IF month > 2 THEN
	count := (month - 1) * 30;
	IF month > 7 THEN count := count + SHR(month - 3,1); ELSE count := count + SHR(month - 4,1); END_IF;
	(* chech for leap year and add one day if true *)
	IF SHL(year,14) = 0 THEN count := count + 1; END_IF;
ELSE
	count := (month - 1) * 31;
END_IF;


SetDataTime := DWORD_TO_DT(DATE_TO_DWORD( DWORD_TO_DATE((INT_TO_DWORD(count + day - 1) + SHR(INT_TO_DWORD(year) * 1461 - 2878169, 2)) * 86400))
				+ INT_TO_DWORD(SECOND)
				+ INT_TO_DWORD(MINUTE) * 60
				+ INT_TO_DWORD(HOUR) * 3600);
END_FUNCTION

(* POU Plant/SYS_Proc, ST *)
PROGRAM SYS_Proc
VAR
	fALARM_PB		:FLT_TAP;
	fALARM_TB		:FLT_TAP;
	fALARM_PM		:FLT_TAP;
	fALARM_ALARM_PM_PB_TB		:FLT_TAP;

(*	fGZB_ST			:FLT_TAP;  (* GATEWAY ZIGBEE *)*)
	fVPN_ST1		:FLT_TAP;  (* VPN CONNECT *)
	fVPN_ST2		:FLT_TAP;  (* VPN STATUS *)
	fKEY_CT_ST		:FLT_TAP;  (* DOOR1 *)
	fKEY_SCT_ST		:FLT_TAP;  (* DOOR2 *)
	fKEY_QE_ST		:FLT_TAP;  (* DOOR3 *)


	fBostAttivo	:FLT_TAP;

	fALARM_MancatoRaggiungimentoAcqua		:FLT_TAP;
	DelayfALARM_MancatoRaggiungimentoAcqua:TON;

	pio: BOOL;
END_VAR
(*************** ISPESL *****************)
(*
fALARM_PB(IN:=ALARM_PB);
IF fALARM_PB.EVH THEN
	LogEv(EL_AlarmStop,EO_PBV,1,1,'Over_Pressure_Alarm');
END_IF

fALARM_TB(IN:=ALARM_TB);
IF fALARM_TB.EVH THEN
	LogEv(EL_AlarmStop,EO_TBV,1,1,'Over_Temperature_Alarm');
END_IF

fALARM_PM(IN:=ALARM_PM);
IF fALARM_PM.EVH THEN
	LogEv(EL_AlarmStop,EO_PMV,1,1,'Under_Pressure_Alarm');
END_IF
*)
(*
fALARM_ALARM_PM_PB_TB(IN:=ALARM_PM_PB_TB);
IF fALARM_ALARM_PM_PB_TB.EVH THEN
	LogEv(EL_AlarmStop,EO_PMV,1,1,'Allarmi_ISPESL');
END_IF
*)

(*



(****************************************)

(*### VPN Connection Check ###*)
fVPN_ST1(IN:=VPN_ST1);
IF fVPN_ST1.EVH THEN
	LogEv(EL_Log,EO_VPN,1,1,'CONNECT_ON');
END_IF
IF fVPN_ST1.EVL THEN
	LogEv(EL_Log,EO_VPN,1,2,'CONNECT_OFF');
END_IF
(*
(*### VPN Status Check ###*)
fVPN_ST2(IN:=VPN_ST2);
IF fVPN_ST2.EVH THEN
	LogEv(EL_Log,EO_VPN,1,3,'STATUS_UP');
END_IF
IF fVPN_ST2.EVL THEN
	LogEv(EL_Wrn,EO_VPN,1,4,'STATUS_DOWN');
END_IF

(*### DOOR01 Status Check ###*)
fKEY_CT_ST(IN:=KEY_CT_ST);
IF fKEY_CT_ST.EVH THEN
	LogEv(EL_Log,EO_DOOR,1,2,'Centrale_termica_Close');
END_IF
IF fKEY_CT_ST.EVL THEN
	LogEv(EL_Wrn,EO_DOOR,1,1,'Centrale_termica_Open');
END_IF

(*### DOOR02 Status Check ###*)
fKEY_SCT_ST(IN:=KEY_SCT_ST);
IF fKEY_SCT_ST.EVH THEN
	LogEv(EL_Log,EO_DOOR,2,2,'Sottocentrale_termica_Close');
END_IF
IF fKEY_SCT_ST.EVL THEN
	LogEv(EL_Wrn,EO_DOOR,2,1,'Sottocentrale_termica_Open');
END_IF
*)
(*### DOOR03 Status Check ###*)
fKEY_QE_ST(IN:=KEY_QE_ST);
IF fKEY_QE_ST.EVH THEN
	LogEv(EL_Log,EO_DOOR,3,2,'Quadro_Close');
END_IF
IF fKEY_QE_ST.EVL THEN
	LogEv(EL_Wrn,EO_DOOR,3,1,'Quadro_Open');
END_IF

*)

pio:=FALSE;
END_PROGRAM

(* POU Utils Functions/FLT_TAP, ST *)
FUNCTION_BLOCK FLT_TAP
VAR_INPUT
	IN		: BOOL;
	TAP		: BYTE:=4;
	INITEV	: BOOL:=TRUE;
END_VAR
VAR_OUTPUT
	OUT		: BOOL;
	EVH		: BOOL;
	EVL		: BOOL;
END_VAR
VAR
	init	: BOOL:=FALSE;
	cnt		: BYTE;
END_VAR
EVH:=FALSE;
EVL:=FALSE;

IF NOT init THEN
	init := TRUE;
	IF INITEV THEN
		OUT  := NOT IN;
		cnt  := TAP;
	ELSE
		OUT  := IN;
	END_IF
END_IF

IF OUT<>IN THEN
	cnt:=cnt+1;
	IF cnt>TAP THEN
		OUT:=IN;
		cnt:=0;
		IF OUT THEN EVH:=TRUE; ELSE EVL:=TRUE; END_IF
	END_IF
ELSE
	cnt:=0;
END_IF
END_FUNCTION_BLOCK

(* POU Utils/USRLED_Update, ST *)
PROGRAM USRLED_Update
VAR
	OldStatus: en_SYS_Status;

	aFS : ARRAY [0..24] OF FLASHING_SEQUENCE :=
		(Colour:=GREEN,  Frequency:=1,   Relation:=128, Duration:=t#0s,    NextIndex:=0),  (* 0 => RUNNING *)
		(Colour:=ORANGE, Frequency:=1,   Relation:=128, Duration:=t#0s,    NextIndex:=1),  (* 1 => INIT *)
		(Colour:=RED,    Frequency:=4,   Relation:=128, Duration:=t#0s,    NextIndex:=2),  (* 2 => ERROR *)
		(Colour:=RED,    Frequency:=10,  Relation:=128, Duration:=t#0s,    NextIndex:=3),  (* 3 => ALARM *)
		(Colour:=ORANGE, Frequency:=200, Relation:=16,  Duration:=t#100ms, NextIndex:=11), (* 10 *)
		(Colour:=ORANGE, Frequency:=200, Relation:=32,  Duration:=t#100ms, NextIndex:=12),
		(Colour:=ORANGE, Frequency:=200, Relation:=64,  Duration:=t#100ms, NextIndex:=13),
		(Colour:=ORANGE, Frequency:=200, Relation:=128, Duration:=t#100ms, NextIndex:=14),
		(Colour:=ORANGE, Frequency:=200, Relation:=192, Duration:=t#100ms, NextIndex:=15),
		(Colour:=ORANGE, Frequency:=200, Relation:=128, Duration:=t#100ms, NextIndex:=16),
		(Colour:=ORANGE, Frequency:=200, Relation:=64,  Duration:=t#100ms, NextIndex:=17),
		(Colour:=ORANGE, Frequency:=200, Relation:=32,  Duration:=t#100ms, NextIndex:=18),
		(Colour:=ORANGE, Frequency:=200, Relation:=16,  Duration:=t#100ms, NextIndex:=19),
		(Colour:=ORANGE, Frequency:=200, Relation:=8,   Duration:=t#100ms, NextIndex:=10),
		(Colour:=GREEN,  Frequency:=200, Relation:=16,  Duration:=t#100ms, NextIndex:=21), (* 20 *)
		(Colour:=GREEN,  Frequency:=200, Relation:=32,  Duration:=t#100ms, NextIndex:=22),
		(Colour:=GREEN,  Frequency:=200, Relation:=64,  Duration:=t#100ms, NextIndex:=23),
		(Colour:=GREEN,  Frequency:=200, Relation:=128, Duration:=t#100ms, NextIndex:=24),
		(Colour:=GREEN,  Frequency:=200, Relation:=192, Duration:=t#100ms, NextIndex:=25),
		(Colour:=GREEN,  Frequency:=200, Relation:=128, Duration:=t#100ms, NextIndex:=26),
		(Colour:=GREEN,  Frequency:=200, Relation:=64,  Duration:=t#100ms, NextIndex:=27),
		(Colour:=GREEN,  Frequency:=200, Relation:=32,  Duration:=t#100ms, NextIndex:=28),
		(Colour:=GREEN,  Frequency:=200, Relation:=16,  Duration:=t#100ms, NextIndex:=29),
		(Colour:=GREEN,  Frequency:=200, Relation:=8,   Duration:=t#100ms, NextIndex:=20);

	pFS : POINTER TO FLASHING_SEQUENCE;


END_VAR
IF Sys.Status <> OldStatus THEN

	OldStatus:=Sys.Status;

	CASE OldStatus OF

		S_STARTUP:
			pFS:=ADR(aFS);
			SET_FLASHING_SEQUENCE(EN:=TRUE, POINTER_TO_POINTER_TO_ARRAY:=ADR(pFS));
			SET_FLASHING_SEQUENCE_INDEX(EN:=TRUE, IMMEDIATE:=FALSE, INDEX:=1);
			START_FLASHING_SEQUENCE(EN:=TRUE);

		S_RUNNING:
			SET_FLASHING_SEQUENCE_INDEX(EN:=TRUE, IMMEDIATE:=TRUE, INDEX:=0);

	END_CASE

END_IF
END_PROGRAM

(* POU Utils Functions/AVERAGE_T, ST *)
FUNCTION_BLOCK AVERAGE_T
VAR_INPUT
	IN: 	INT;
END_VAR
VAR_OUTPUT
	HI:		INT;
	AVG:	INT;
	LOW:	INT;
	ERR:	BOOL;
END_VAR
VAR
	sum:	DINT;
	cnt:	WORD;
END_VAR
IF cnt>=65000 THEN
	ERR:=TRUE;
	Read();
	sum := sum - AVG;
	cnt := cnt + 1;
END_IF

sum := sum + IN;
cnt := cnt + 1;

IF IN<LOW THEN  LOW:=IN; END_IF
IF IN>HI  THEN HI :=IN; END_IF
END_FUNCTION_BLOCK
ACTION Read:
AVG := DINT_TO_INT(sum/cnt);
END_ACTION
ACTION Reset:
HI:=IN;
AVG:=IN;
LOW:=IN;
ERR:=FALSE;

sum:=IN;
cnt:=1;
END_ACTION

(* POU Utils Functions/COPY_32SWAP16, ST *)
FUNCTION COPY_32SWAP16:BOOL
VAR_INPUT
	pSourceAddress		:POINTER TO ARRAY[1..2] OF WORD;
	pDestinationAddress	:POINTER TO ARRAY[1..2] OF WORD;
END_VAR
VAR
END_VAR
pDestinationAddress^[1]:=pSourceAddress^[2];
pDestinationAddress^[2]:=pSourceAddress^[1];
END_FUNCTION

(* POU Utils Functions/FLT_EVENT, ST *)
FUNCTION_BLOCK FLT_EVENT
VAR_INPUT
	IN		: BOOL;
	INITEV	: BOOL:=TRUE;
END_VAR
VAR_OUTPUT
	EVH		: BOOL;
	EVL		: BOOL;
END_VAR
VAR
	init	: BOOL:=FALSE;
	old		: BOOL;
END_VAR
EVH:=FALSE;
EVL:=FALSE;

IF NOT init THEN
	init:=TRUE;
	IF INITEV THEN
		old := NOT IN;
	ELSE
		old := IN;
	END_IF
END_IF

IF old<>IN THEN
	old:=IN;
	IF IN THEN EVH:=TRUE; ELSE EVL:=TRUE; END_IF
END_IF
END_FUNCTION_BLOCK

(* POU Utils Functions/FLT_TIME, ST *)
FUNCTION_BLOCK FLT_TIME
VAR_INPUT
	IN		: BOOL;
	TTAP	: TIME:=T#5s;
	INITEV	: BOOL:=TRUE;
END_VAR
VAR_OUTPUT
	OUT		: BOOL;
	EVH		: BOOL;
	EVL		: BOOL;
END_VAR
VAR
	init	: BOOL:=FALSE;
	timer	: TON;
END_VAR
EVH:=FALSE;
EVL:=FALSE;

IF NOT init THEN
	init := TRUE;
	IF INITEV THEN
		OUT  := NOT IN;
	ELSE
		OUT  := IN;
	END_IF
END_IF

IF OUT<>IN THEN
	timer(IN:=TRUE,PT:=TTAP);
	IF timer.Q THEN
		OUT:=IN;
		timer(IN:=FALSE);
		IF OUT THEN EVH:=TRUE; ELSE EVL:=TRUE; END_IF
	END_IF
ELSE
	timer(IN:=FALSE);
END_IF
END_FUNCTION_BLOCK

(* POU Utils Functions/FUN_2Word_to_REAL, ST *)
FUNCTION FUN_2Word_to_REAL : REAL
VAR_INPUT

	WORDH:WORD;
	WORDL:WORD;
	Decimali:INT;
	signed:BOOL;     (* false unsigned - true signed *)

END_VAR

VAR

	ValoreDWord: DWORD;
	ValoreDint: DINT;
	testINT1: DINT;
	testINT2: DINT;


END_VAR
IF signed THEN

		(* Stabilisco il segno della variabile letta *)

		IF WORDH> 16#8000 THEN
			ValoreDint:=((16#FFFFFFFF-(WORDH*65535+WORDL)))*(-1);
		ELSE
			ValoreDint:=(WORDH*65535+WORDL);
		END_IF;

	CASE Decimali OF
		0 : FUN_2Word_to_REAL:=DINT_TO_REAL (ValoreDint);
		1 : FUN_2Word_to_REAL:=DINT_TO_REAL (ValoreDint)/10;
		2 : FUN_2Word_to_REAL:=DINT_TO_REAL (ValoreDint)/100;
		3 : FUN_2Word_to_REAL:=DINT_TO_REAL (ValoreDint)/1000;
		4 : FUN_2Word_to_REAL:=DINT_TO_REAL (ValoreDint)/10000;
		5 : FUN_2Word_to_REAL:=DINT_TO_REAL (ValoreDint)/100000;
		6 : FUN_2Word_to_REAL:=DINT_TO_REAL (ValoreDint)/1000000;
	END_CASE;


ELSE
	ValoreDWord:=(WORDH*65535+WORDL);

	CASE Decimali OF
		0 : FUN_2Word_to_REAL:=DWORD_TO_REAL (ValoreDWord);
		1 : FUN_2Word_to_REAL:=DWORD_TO_REAL (ValoreDWord)/10;
		2 : FUN_2Word_to_REAL:=DWORD_TO_REAL (ValoreDWord)/100;
		3 : FUN_2Word_to_REAL:=DWORD_TO_REAL (ValoreDWord)/1000;
		4 : FUN_2Word_to_REAL:=DWORD_TO_REAL (ValoreDWord)/10000;
		5 : FUN_2Word_to_REAL:=DWORD_TO_REAL (ValoreDWord)/100000;
		6 : FUN_2Word_to_REAL:=DWORD_TO_REAL (ValoreDWord)/1000000;
	END_CASE;
END_IF;
END_FUNCTION

(* POU Utils/FUN_ByteAsci, ST *)
FUNCTION FUN_ByteAsci : STRING(1)
VAR_INPUT
	ByteIn:BYTE;
END_VAR
VAR
END_VAR
CASE ByteIn OF

	32: FUN_ByteAsci:=' ';
	33: FUN_ByteAsci:='!';
	34: FUN_ByteAsci:='"';
	35: FUN_ByteAsci:='#';

	37: FUN_ByteAsci:='%';
	38: FUN_ByteAsci:='&';

	40: FUN_ByteAsci:='(';
	41: FUN_ByteAsci:=')';
	42: FUN_ByteAsci:='*';
	43: FUN_ByteAsci:='+';
	44: FUN_ByteAsci:=',';
	45: FUN_ByteAsci:='-';
	46: FUN_ByteAsci:='.';
	47: FUN_ByteAsci:='/';
	48: FUN_ByteAsci:='0';
	49: FUN_ByteAsci:='1';
	50: FUN_ByteAsci:='2';
	51: FUN_ByteAsci:='3';
	52: FUN_ByteAsci:='4';
	53: FUN_ByteAsci:='5';
	54: FUN_ByteAsci:='6';
	55: FUN_ByteAsci:='7';
	56: FUN_ByteAsci:='8';
	57: FUN_ByteAsci:='9';
	58: FUN_ByteAsci:=':';
	59: FUN_ByteAsci:=';';
	60: FUN_ByteAsci:='<';
	61: FUN_ByteAsci:='=';
	62: FUN_ByteAsci:='>';
	63: FUN_ByteAsci:='?';
	64: FUN_ByteAsci:='@';
	65: FUN_ByteAsci:='A';
	66: FUN_ByteAsci:='B';
	67: FUN_ByteAsci:='C';
	68: FUN_ByteAsci:='D';
	69: FUN_ByteAsci:='E';
	70: FUN_ByteAsci:='F';
	71: FUN_ByteAsci:='G';
	72: FUN_ByteAsci:='H';
	73: FUN_ByteAsci:='I';
	74: FUN_ByteAsci:='J';
	75: FUN_ByteAsci:='K';
	76: FUN_ByteAsci:='L';
	77: FUN_ByteAsci:='M';
	78: FUN_ByteAsci:='N';
	79: FUN_ByteAsci:='O';
	80: FUN_ByteAsci:='P';
	81: FUN_ByteAsci:='Q';
	82: FUN_ByteAsci:='R';
	83: FUN_ByteAsci:='S';
	84: FUN_ByteAsci:='T';
	85: FUN_ByteAsci:='U';
	86: FUN_ByteAsci:='V';
	87: FUN_ByteAsci:='W';
	88: FUN_ByteAsci:='X';
	89: FUN_ByteAsci:='Y';
	90: FUN_ByteAsci:='Z';
	91: FUN_ByteAsci:='[';
	92: FUN_ByteAsci:='\';
	93: FUN_ByteAsci:=']';
	94: FUN_ByteAsci:='^';
	95: FUN_ByteAsci:='_';
	96: FUN_ByteAsci:='`';
	97: FUN_ByteAsci:='a';
	98: FUN_ByteAsci:='b';
	99: FUN_ByteAsci:='c';
	100: FUN_ByteAsci:='d';
	101: FUN_ByteAsci:='e';
	102: FUN_ByteAsci:='f';
	103: FUN_ByteAsci:='g';
	104: FUN_ByteAsci:='h';
	105: FUN_ByteAsci:='i';
	106: FUN_ByteAsci:='j';
	107: FUN_ByteAsci:='k';
	108: FUN_ByteAsci:='l';
	109: FUN_ByteAsci:='m';
	110: FUN_ByteAsci:='n';
	111: FUN_ByteAsci:='o';
	112: FUN_ByteAsci:='p';
	113: FUN_ByteAsci:='q';
	114: FUN_ByteAsci:='r';
	115: FUN_ByteAsci:='s';
	116: FUN_ByteAsci:='t';
	117: FUN_ByteAsci:='u';
	118: FUN_ByteAsci:='v';
	119: FUN_ByteAsci:='w';
	120: FUN_ByteAsci:='x';
	121: FUN_ByteAsci:='y';
	122: FUN_ByteAsci:='z';
	123: FUN_ByteAsci:='{';
	124: FUN_ByteAsci:='|';
	125: FUN_ByteAsci:='}';
	126: FUN_ByteAsci:='~';

	167: FUN_ByteAsci:='°';
	176: FUN_ByteAsci:='°';


ELSE
	FUN_ByteAsci:='';

END_CASE
END_FUNCTION

(* POU Utils Functions/FUN_DEAD_ZONE, ST *)
FUNCTION FUN_DEAD_ZONE : INT
VAR_INPUT
	X : INT;
	L : INT;
END_VAR
VAR
	DEAD_BAND: BOOL;
END_VAR
IF X>=FUN_DEAD_ZONE+L THEN
	FUN_DEAD_ZONE := X ;
ELSIF X <= FUN_DEAD_ZONE-L THEN
	FUN_DEAD_ZONE := X;
ELSE
	FUN_DEAD_ZONE :=FUN_DEAD_ZONE;
END_IF;
END_FUNCTION

(* POU Utils Functions/LAMP_AL_GENERALE, ST *)
FUNCTION_BLOCK LAMP_AL_GENERALE
VAR_INPUT

	Allarme: BOOL;
	Warning: BOOL;
END_VAR
VAR_OUTPUT
	SistemaOK:BOOL;
	SistemaInAllarme:BOOL;
	SistemaWarning:BOOL;
	AllarmeLampada:BOOL;
END_VAR
VAR
	Lampeggio:BLINK;
END_VAR
IF Allarme THEN       					(* Se Allarme Attivo Lucde fissa ON *)
	SistemaInAllarme:=TRUE;
	SistemaWarning:=FALSE;
	AllarmeLampada:=TRUE;
ELSIF Warning THEN					(* Se Allarme Attivo Lucde fissa pulse *)
	SistemaInAllarme:=FALSE;
	SistemaWarning:=TRUE;
	Lampeggio(ENABLE:=TRUE , TIMELOW:=t#1s , TIMEHIGH:=t#1s , OUT=>AllarmeLampada );
ELSE
	SistemaInAllarme:=FALSE;
	SistemaWarning:=FALSE;
	AllarmeLampada:=FALSE;
END_IF
END_FUNCTION_BLOCK

(* POU Utils Functions/LINEAR_BAD, ST *)
FUNCTION LINEAR_BAD : INT (* Linear interpolation *)
VAR_INPUT
	PuntoMinX	: INT;
	PuntoMaxX	: INT;
	ValIn		: INT;
	PuntoMinY	: REAL;
	PuntoMaxY	: REAL;
	Decimali	: BYTE;
END_VAR
VAR
	Gain				: REAL;
	PuntoMinX_R			: REAL;
	PuntoMaxX_R			: REAL;
	Linearizzazione_R	: REAL;
END_VAR
PuntoMinX_R:=INT_TO_REAL(PuntoMinX);
PuntoMaxX_R:=INT_TO_REAL(PuntoMaxX);

Gain:=(PuntoMaxX_R-PuntoMinX_R)/(PuntoMaxY-PuntoMinY);	(* Calcolo in guadagno per la linarizzazione *)
Linearizzazione_R:=PuntoMinx+(Gain*(ValIn-PuntoMinY));	(* Ottengo il valore linearizzato *)

LINEAR_BAD:=REAL_TO_INT(Linearizzazione_R*(EXPT(10, Decimali)));  (* Ottengo intero con i decimai voluti *)
END_FUNCTION

(* POU Utils Functions/MEMCLR, ST *)
FUNCTION MEMCLR:BOOL
VAR_INPUT
	pDestinationAddress:POINTER TO ARRAY[1..2] OF BYTE;
	BytesToClear:WORD;
END_VAR
VAR
END_VAR
WHILE (BytesToClear > 0) DO
	pDestinationAddress^[1]:=0;
	pDestinationAddress:=ADR(pDestinationAddress^[2]); (* increment destination *)
	BytesToClear:=BytesToClear -1; (* decrement number of bytes to copy *)
END_WHILE
END_FUNCTION

(* POU Plant_Objects/obj_AI_GEN, ST *)
FUNCTION_BLOCK obj_AI_GEN
(* === TEMPERATURE PROBE FROM ANALOG INPUT ===
   v1.0[16/04/05] - Versioning
*)
VAR_INPUT
	(* Settings *)
	ID				: BYTE;
	PuntoMinX		: INT;			(* Parametri per la scalatura *)
	PuntoMaxX		: INT;
	PuntoMinY		: REAL;
	PuntoMaxY		: REAL;
	Decimali		: BYTE:=1;
	SogliaHH		: WORD;			(* Soglia per segnalazione Allarme Extra Range in alto - Solitamente sondo in CC *)
	SogliaHL		: WORD;			(* Soglia per segnalazione Allarme Extra Range in Basso - Solitamente sondo Aperta *)
	SogliaWH		: REAL;			(* Soglia per segnalazione Warning  in alto  *)
	SogliaWL		: REAL;    		(* Soglia per segnalazione Warning in basso  *)
	TAP				: INT:=2000;	(* Filtro in msec *)
	INITEV			: BOOL:= TRUE;	(* Generate init OK event *)
	(* Physical input *)
	AI_INPUT		: WORD;    		(* Sensor analog input *)
	TipoSensore:STRING(12);
END_VAR
VAR_OUTPUT
	WRN				: BOOL;	(* Segnalazione Warning *)
	ERR				: BOOL; (* Segnalazione Errore *)
	ValoreScalato	: INT;
	(* Status *)
	Status_Log	: BYTE;
	Status_Vis 	: DWORD;
END_VAR
VAR
	SegnaleHH	: BOOL;
	SegnaleHL	: BOOL;
	SegnaleOK	: BOOL;
	SegnaleWH	: BOOL;
	SegnaleWL	: BOOL;
    FiltroWRN	: TON;
    FiltroOK	: TON;
    FiltroERR	: TON;
END_VAR
(* Verifico che le variabile letta dall'ingresso Analogico  sia dentro i range
ATTENZIONE I LIMITI SPESSO SONO IN WORD VERIFICA  TABELLA MANUALE WAGO  *)

SegnaleHH:=(AI_INPUT>=SogliaHH);
SegnaleHL:=(AI_INPUT<=SogliaHL);
SegnaleOK:=NOT (SegnaleHH OR SegnaleHL);

(* Linerarizzo il segnale di ingresso e la converto in unita ingegneristiche *)
ValoreScalato:=LINEAR_BAD(PuntoMinX, PuntoMaxX, AI_INPUT, PuntoMinY, PuntoMaxY, Decimali);


IF SegnaleOK  THEN
	(*  Verifica  e segnalazione Warning *)
	SegnaleWH:=(ValoreScalato>SogliaWH*(EXPT(10, Decimali)));
	SegnaleWL:=(ValoreScalato<SogliaWL*(EXPT(10, Decimali)));

	Status_Log:=0;
	Status_Vis:=16#20F020;    (* Indicazione WEB Visu Sonda OK *)

	FiltroWRN( IN:=(SegnaleWH OR SegnaleWL), PT:=INT_TO_TIME(TAP) );    (* Filtro su LOG *)
	IF  FiltroWRN.Q THEN     (* Condizione di WARNING *)
		IF NOT WRN THEN
			WRN:=TRUE;
			Status_Log:=1;
			LogEv(EL_Wrn,EO_ZTHL,ID,SEL(ValoreScalato<=SogliaWL,3,2),INT_TO_STRING(ValoreScalato));
		END_IF
	END_IF

    IF (INITEV OR WRN OR ERR) AND NOT FiltroWRN.Q THEN
		FiltroWRN(IN:=FALSE  , PT:=INT_TO_TIME(TAP));    (* Resetto il Filtro su LOG WRN  *)
		FiltroERR(IN:=FALSE  , PT:=INT_TO_TIME(TAP));    (* Resetto il Filtro su LOG ERR *)
		INITEV:=FALSE; ERR:=FALSE; WRN:=FALSE;
		LogEv(EL_Log,EO_ZTHL,ID,1,'');
	END_IF
ELSE
	FiltroERR(IN:=TRUE  , PT:= INT_TO_TIME(TAP) );    (* Filtro su LOG *)
	IF  FiltroERR.Q THEN     (* Condizione di WARNING *)
		IF NOT ERR THEN
			ERR:=TRUE;
			Status_Log:=2;

			IF SegnaleHH THEN LogEv(EL_Alarm,EO_ZTHL,ID,6,INT_TO_STRING(ValoreScalato));END_IF;
			IF SegnaleHL THEN LogEv(EL_Alarm,EO_ZTHL,ID,4,INT_TO_STRING(ValoreScalato));END_IF;
		END_IF
	END_IF

	Status_Vis:=16#2020F0;   (* Indicazione WEB Visu Sonda KO *)
END_IF



(* Status Log *)
IF ERR THEN
	Status_Log := 2;
	Status_Vis := COLOR_RED;
ELSIF WRN THEN
	Status_Log := 1;
	Status_Vis := COLOR_YELLOW;
ELSE
	Status_Log := 0; Status_Vis := COLOR_GREEN;
END_IF
END_FUNCTION_BLOCK
ACTION AddLogData:
Logger.s1:=CONCAT('&',TipoSensore);
IF ID<10 THEN Logger.s1:=CONCAT(Logger.s1,'0');END_IF
Logger.s1:=CONCAT(Logger.s1,BYTE_TO_STRING(ID));
Logger.s1:=CONCAT(Logger.s1,'=');


Logger.s1:=CONCAT(Logger.s1,BYTE_TO_STRING(0));     (* OUT_LQI*)
Logger.s1:=CONCAT(Logger.s1,';');
Logger.s1:=CONCAT(Logger.s1,INT_TO_STRING(0 ));		(* OUT_TEMP*)
Logger.s1:=CONCAT(Logger.s1,';');
Logger.s1:=CONCAT(Logger.s1,INT_TO_STRING(0 ));		(* OUT_HYGRO*)
Logger.s1:=CONCAT(Logger.s1,';');
Logger.s1:=CONCAT(Logger.s1,INT_TO_STRING(ValoreScalato));		(* OUT_LUX*)
Logger.s1:=CONCAT(Logger.s1,';');
Logger.s1:=CONCAT(Logger.s1,INT_TO_STRING(0));				(* OUT_VBATT*)
Logger.s1:=CONCAT(Logger.s1,';');

Logger.s1:=CONCAT(Logger.s1,BYTE_TO_STRING(Status_Log));
ADDSTRING(ADR(Logger.TData), ADR(Logger.s1), Logger.TLen);
END_ACTION

(* POU Plant_Objects/obj_Anz_Lovato_ETH, ST *)
FUNCTION_BLOCK obj_Anz_Lovato_ETH
(* === MODBUS-TCP PROTOCOL INTERFACE ===
   v1.0[10/06/15] - Create
*)
VAR CONSTANT
	VARS_Max	: BYTE := 32;
END_VAR
VAR_INPUT
	(* Settings *)
	ID			: BYTE;
	IP			: STRING;
	PORT		: WORD:=502;
	(* Interface *)
	MB_MASTER	: ETHERNET_MODBUSMASTER_TCP;
	MB_READBUF	: ARRAY [0..128] OF WORD;
	MB_WRITEBUF : ARRAY [0..128] OF WORD;
	MB_Start	: BOOL;
	MB_Lock		: BOOL;
	(* Variables management *)
	VARS_En		: BOOL;
	VARS		: ARRAY [0..VARS_Max] OF typ_MODBUS_VAR;
	VARS_Check	: BOOL;
	VARS_Alarm	: BOOL;
	(* Variables allocation *)
	VAR_Pointer : POINTER TO ARRAY[0..99] OF WORD;
	VAR_Cfg		: POINTER TO typ_MODBUS_VAR;

	(* Type of ANZ: 1-phase or 3-phase *)
	contabilizerMode:BYTE:=1;







END_VAR
VAR_OUTPUT

	(* output records representing the data in according to the ANZ Clevergy Web format *)
	measures						: typ_ANZ_real;

	(* Status *)
	Status_Log	: BYTE;
	Status_Vis	: DWORD;
END_VAR
VAR
	sta         : BYTE :=0;
	i			: BYTE;
	j			: BYTE;
	Alarm		: FLT_EVENT;

	VarTmr		: TON := (PT:=T#1s);
	VarSta		: BYTE; (* Status *)
	VarCnt		: BYTE; (* Scan counter *)
	VarRetry	: BYTE;
	VarAlarm	: BYTE; (* Last variable with errors *)


	state : INT;
	ReadTmr		:	TON := (PT:=T#5s);
	retry		:	BYTE;
	retryErr	:	BYTE;
	retryErrMax	:	BYTE := 2;
	ErroreComuModBus: BOOL;
	fModbusAlr:BOOL;

	MB_RegistriHoldingLetti: ARRAY [0..80] OF WORD;

	x: INT;

	(* da diego per gestione stato stringa > 255*)
	temp :STRING(255);
	tempRaw		: ARRAY [0..MAX_SEND_TCP_CLIENT] OF BYTE;
	tempRawLen :DINT;
	longString:STRING(300);


	TimeOutModBus: TON;
	ErroreTimeOut: BOOL;
	test_moreno: BOOL;
	test_moreno1: WORD;
	test_moreno2: BYTE;
	AppoggioDWORD: DWORD;



	testindirizzo:INT;
	testNumeroIndirizzo:INT;


	testR1: REAL;
	testR2: REAL;
	testR3: REAL;
	testR4: REAL;
	testR5: REAL;




END_VAR
CASE state OF
	0:	(* Refresh time manager *)
		ReadTmr(IN:=NOT ReadTmr.Q,pt:=t#1000ms);
			MB_Start:=FALSE;

		(*A tempo interrogo il nodo sempre che non ci sia qualcuno che lo sta interrogando in quel momento *)
		IF  ReadTmr.Q THEN
			state := 5;
		END_IF
	5:
	test_moreno:=MB_MASTER.xIS_CONNECTED;
	test_moreno1:=MB_MASTER.wERROR;
	test_moreno2:=MB_MASTER.bRESPONSE_UNIT_ID;
		IF  MB_MASTER.xIS_CONNECTED THEN
			state :=10;
		END_IF
	(**** Leggo le Analogiche a Disposzione  ****)

	10:	(* richiedo lettura Holding Registere   *)

			MB_MASTER.bUNIT_ID := 1;
			MB_MASTER.bFUNCTION_CODE:=3;
			MB_MASTER.wREAD_ADDRESS:=1;
			MB_MASTER.wREAD_QUANTITY:=72;
			MB_Start:=TRUE;
			state := 20;


	20:	(* Risposta all'interrogazione *)
		IF NOT MB_Start THEN
			IF MB_MASTER.wERROR<>MB_NO_ERROR THEN
				state:=300;
			ELSE

				FOR x:=0 TO MB_MASTER.wREAD_QUANTITY DO
					MB_RegistriHoldingLetti[x+MB_MASTER.wREAD_ADDRESS] := MB_READBUF[x];
				END_FOR

				state := 30;

			END_IF
		END_IF

	30:	(* Risposta all'interrogazione *)
		IF NOT MB_Start THEN
			IF MB_MASTER.wERROR<>MB_NO_ERROR THEN
				state:=300;
			ELSE




			(* voltages *)
			measures.V_L1N:=FUN_2Word_to_REAL(MB_RegistriHoldingLetti[1],MB_RegistriHoldingLetti[2],2,FALSE);
			measures.V_L2N:=FUN_2Word_to_REAL(MB_RegistriHoldingLetti[3],MB_RegistriHoldingLetti[4],2,FALSE);
			measures.V_L3N:=FUN_2Word_to_REAL(MB_RegistriHoldingLetti[5],MB_RegistriHoldingLetti[6],2,FALSE);
			measures.V_L1L2:=FUN_2Word_to_REAL(MB_RegistriHoldingLetti[13],MB_RegistriHoldingLetti[14],2,FALSE);
			measures.V_L2L3:=FUN_2Word_to_REAL(MB_RegistriHoldingLetti[15],MB_RegistriHoldingLetti[16],2,FALSE);
			measures.V_L3L1:=FUN_2Word_to_REAL(MB_RegistriHoldingLetti[17],MB_RegistriHoldingLetti[18],2,FALSE);
			(* frequency *)
			measures.FREQ:=(FUN_2Word_to_REAL(MB_RegistriHoldingLetti[49],MB_RegistriHoldingLetti[50],2,FALSE));

			(* currents *)
			measures.I_L1:=FUN_2Word_to_REAL(MB_RegistriHoldingLetti[7],MB_RegistriHoldingLetti[8],4,FALSE);
			measures.I_L2:=FUN_2Word_to_REAL(MB_RegistriHoldingLetti[9],MB_RegistriHoldingLetti[10],4,FALSE);
			measures.I_L3:=FUN_2Word_to_REAL(MB_RegistriHoldingLetti[11],MB_RegistriHoldingLetti[12],4,FALSE);

			measures.I_L1_Max:=FUN_2Word_to_REAL(MB_RegistriHoldingLetti[7],MB_RegistriHoldingLetti[8],4,FALSE);
			measures.I_L2_Max:=FUN_2Word_to_REAL(MB_RegistriHoldingLetti[9],MB_RegistriHoldingLetti[10],4,FALSE);
			measures.I_L3_Max:=FUN_2Word_to_REAL(MB_RegistriHoldingLetti[11],MB_RegistriHoldingLetti[12],4,FALSE);

			(* power factors *)
			measures.PF_L1:=FUN_2Word_to_REAL(MB_RegistriHoldingLetti[37],MB_RegistriHoldingLetti[38],4,TRUE);
			measures.PF_L2:=FUN_2Word_to_REAL(MB_RegistriHoldingLetti[39],MB_RegistriHoldingLetti[40],4,TRUE);
			measures.PF_L3:=FUN_2Word_to_REAL(MB_RegistriHoldingLetti[41],MB_RegistriHoldingLetti[42],4,TRUE);

			(* active powers *)
			measures.P_3P	:=FUN_2Word_to_REAL(MB_RegistriHoldingLetti[57],MB_RegistriHoldingLetti[58],2,TRUE);
			measures.P_3P_Avg:=FUN_2Word_to_REAL(MB_RegistriHoldingLetti[57],MB_RegistriHoldingLetti[58],2,TRUE);
			measures.P_3P_Max:=0;

			(* reactive powers *)
			measures.Q_3P	:=FUN_2Word_to_REAL(MB_RegistriHoldingLetti[59],MB_RegistriHoldingLetti[60],2,TRUE);
			measures.Q_3P_Max:=0;	(* VAr *)

			(* active energy *)
			measures.WH_3P:=0;

			(* reactive energy *)
			measures.VARH_3P:=0;

			(* cosphi *)
			measures.COSPHI_L1:=FUN_2Word_to_REAL(MB_RegistriHoldingLetti[43],MB_RegistriHoldingLetti[44],4,TRUE);
			measures.COSPHI_L2:=FUN_2Word_to_REAL(MB_RegistriHoldingLetti[45],MB_RegistriHoldingLetti[46],4,TRUE);
			measures.COSPHI_L3:=FUN_2Word_to_REAL(MB_RegistriHoldingLetti[47],MB_RegistriHoldingLetti[48],4,TRUE);




				state := 295;

			END_IF
		END_IF









	40:	(* richiedo lettura Holding Registere   *)

			MB_MASTER.bUNIT_ID := 1;
			MB_MASTER.bFUNCTION_CODE:=3;
			MB_MASTER.wREAD_ADDRESS:=6687;
			MB_MASTER.wREAD_QUANTITY:=10;
			MB_Start:=TRUE;
			state := 50;


	50:	(* Risposta all'interrogazione *)
		IF NOT MB_Start THEN
			IF MB_MASTER.wERROR<>MB_NO_ERROR THEN
				state:=300;
			ELSE

			(* active energy *)
			measures.WH_3P:=FUN_2Word_to_REAL(MB_READBUF[1],MB_READBUF[2],2,FALSE);   (* kwh *)

			(* reactive energy *)
			measures.VARH_3P:=FUN_2Word_to_REAL(MB_READBUF[5],MB_READBUF[6],2,FALSE);   (* kVarh *)


			testR1:=FUN_2Word_to_REAL(MB_READBUF[1],MB_READBUF[2],2,FALSE);
			testR2:=FUN_2Word_to_REAL(MB_READBUF[3],MB_READBUF[4],2,FALSE);
			testR3:=FUN_2Word_to_REAL(MB_READBUF[5],MB_READBUF[6],2,FALSE);
			testR4:=FUN_2Word_to_REAL(MB_READBUF[7],MB_READBUF[8],2,FALSE);
			testR5:=FUN_2Word_to_REAL(MB_READBUF[9],MB_READBUF[10],2,FALSE);







			state := 295;

			END_IF
		END_IF





		295:
		IF NOT MB_Start THEN
			IF  MB_MASTER.wERROR<>MB_NO_ERROR THEN (*OR ModBus.MB_MASTER.MB_Error<>0 THEN*)
				state := 300;
			ELSE
				retryErr := 0;
				retry := 0;
				state := 0;
					IF ErroreComuModBus=TRUE THEN
						LogEv(EL_Log,EO_MODBUS_TCP,ID,2,'Comunicazione_ristabilita');
						ErroreComuModBus := FALSE;
						fModbusAlr := FALSE;

				(*	WarningCtr := SEL(WarningCtr=0, WarningCtr-1, 0); *)
					END_IF
			END_IF
		END_IF



	(**** CHECK MODBUS ERROR ****)
	300: 	(* Release MODBUS *)
			retry:=retry+1;
			IF retry>3 THEN
				retry:=0;

				(* Verify if slave is dead *)
				IF retryErr < retryErrMaX THEN
					retryErr := retryErr + 1;
				ELSE
					fModbusAlr := TRUE;
					(* Verify ModBus error	*)

					IF fModbusAlr AND ErroreComuModBus=FALSE THEN
						LogEv(SEL(MB_MASTER.wERROR>0,EL_Wrn,EL_Alarm),EO_MODBUS_TCP,ID,1,WORD_TO_STRING(MB_MASTER.wERROR));
						ErroreComuModBus := TRUE;
					END_IF
				END_IF

				END_IF
			state:=0;
END_CASE



MB_MASTER( strIP_ADDRESS:=IP, wPORT:=PORT, tTIME_OUT:=T#750MS, (*xCONNECT:=TRUE,*)
		   ptREAD_DATA:=ADR(MB_READBUF), ptSEND_DATA:=ADR(MB_WRITEBUF), xSEND:=MB_Start );

IF state<>0 THEN
	MB_MASTER.xCONNECT:=TRUE;
ELSE
	MB_MASTER.xCONNECT:=FALSE;
END_IF
(*
(* Process variable management *)
IF VARS_En THEN VARS_Process(); END_IF
*)

(* Controllo Time Out Ciclo ModBus *)

TimeOutModBus(In:=state<>0,PT:=t#5s);
IF TimeOutModBus.Q THEN
	State:=300;
END_IF


(* Log/visu status *)
   IF Alarm.IN   THEN Status_Log:=2; Status_Vis:=COLOR_RED;
ELSIF Vars_Alarm OR ErroreComuModBus  THEN
	Status_Log:=1; Status_Vis:=COLOR_YELLOW;
  ELSE
	Status_Log:=0; Status_Vis:=COLOR_GREEN;
END_IF
END_FUNCTION_BLOCK
ACTION AddLogData:
Logger.s1:=INSERT('&ANZ=',WORD_TO_STRING(ID),4);
IF ID<10 THEN Logger.s1:=INSERT(Logger.s1,'0',4); END_IF

Logger.s1:=CONCAT(Logger.s1,REAL_TO_STRING(measures.V_L1N));		Logger.s1:=CONCAT(Logger.s1,';');
Logger.s1:=CONCAT(Logger.s1,REAL_TO_STRING(measures.V_L2N));		Logger.s1:=CONCAT(Logger.s1,';');
Logger.s1:=CONCAT(Logger.s1,REAL_TO_STRING(measures.V_L3N));		Logger.s1:=CONCAT(Logger.s1,';');
Logger.s1:=CONCAT(Logger.s1,REAL_TO_STRING(measures.V_L1L2));		Logger.s1:=CONCAT(Logger.s1,';');
Logger.s1:=CONCAT(Logger.s1,REAL_TO_STRING(measures.V_L2L3));		Logger.s1:=CONCAT(Logger.s1,';');
Logger.s1:=CONCAT(Logger.s1,REAL_TO_STRING(measures.V_L3L1));		Logger.s1:=CONCAT(Logger.s1,';');

Logger.s1:=CONCAT(Logger.s1,REAL_TO_STRING(measures.FREQ*100));		Logger.s1:=CONCAT(Logger.s1,';');

Logger.s1:=CONCAT(Logger.s1,REAL_TO_STRING(measures.I_L1));		Logger.s1:=CONCAT(Logger.s1,';');
Logger.s1:=CONCAT(Logger.s1,REAL_TO_STRING(measures.I_L2));		Logger.s1:=CONCAT(Logger.s1,';');
Logger.s1:=CONCAT(Logger.s1,REAL_TO_STRING(measures.I_L3));		Logger.s1:=CONCAT(Logger.s1,';');
Logger.s1:=CONCAT(Logger.s1,REAL_TO_STRING(measures.I_L1_Max)); 	Logger.s1:=CONCAT(Logger.s1,';');
Logger.s1:=CONCAT(Logger.s1,REAL_TO_STRING(measures.I_L2_Max)); 	Logger.s1:=CONCAT(Logger.s1,';');
Logger.s1:=CONCAT(Logger.s1,REAL_TO_STRING(measures.I_L3_Max)); 	Logger.s1:=CONCAT(Logger.s1,';');

Logger.s1:=CONCAT(Logger.s1,REAL_TO_STRING(measures.PF_L1));		Logger.s1:=CONCAT(Logger.s1,';');
Logger.s1:=CONCAT(Logger.s1,REAL_TO_STRING(measures.PF_L2));		Logger.s1:=CONCAT(Logger.s1,';');
Logger.s1:=CONCAT(Logger.s1,REAL_TO_STRING(measures.PF_L3));		Logger.s1:=CONCAT(Logger.s1,';');

Logger.s1:=CONCAT(Logger.s1,REAL_TO_STRING(measures.P_3P));		Logger.s1:=CONCAT(Logger.s1,';');
Logger.s1:=CONCAT(Logger.s1,REAL_TO_STRING(measures.P_3P_Avg)); 	Logger.s1:=CONCAT(Logger.s1,';');
Logger.s1:=CONCAT(Logger.s1,REAL_TO_STRING(measures.P_3P_Max)); 	Logger.s1:=CONCAT(Logger.s1,';');

Logger.s1:=CONCAT(Logger.s1,REAL_TO_STRING(measures.Q_3P));			Logger.s1:=CONCAT(Logger.s1,';');
Logger.s1:=CONCAT(Logger.s1, REAL_TO_STRING(measures.Q_3P_Max));		Logger.s1:=CONCAT(Logger.s1,';');

Logger.s1:=CONCAT(Logger.s1,REAL_TO_STRING(measures.WH_3P*100));			Logger.s1:=CONCAT(Logger.s1,';');
Logger.s1:=CONCAT(Logger.s1,REAL_TO_STRING(measures.VARH_3P*100));			Logger.s1:=CONCAT(Logger.s1,';');

Logger.s1:=CONCAT(Logger.s1,BYTE_TO_STRING(Status_Log)); 					Logger.s1:=CONCAT(Logger.s1,';');

Logger.s1:=CONCAT(Logger.s1,REAL_TO_STRING(measures.COSPHI_L1));		Logger.s1:=CONCAT(Logger.s1,';');
Logger.s1:=CONCAT(Logger.s1,REAL_TO_STRING(measures.COSPHI_L2));		Logger.s1:=CONCAT(Logger.s1,';');
Logger.s1:=CONCAT(Logger.s1,REAL_TO_STRING(measures.COSPHI_L3));		Logger.s1:=CONCAT(Logger.s1,';');

Logger.s1:=CONCAT(Logger.s1,BYTE_TO_STRING(contabilizerMode));

ADDSTRING(ADR(Logger.TData), ADR(Logger.s1), Logger.TLen);
END_ACTION

(* POU Plant_Objects/obj_Anz_Seneca_ETH, ST *)
FUNCTION_BLOCK obj_Anz_Seneca_ETH
(* === MODBUS-TCP PROTOCOL INTERFACE ===
   v1.0[10/06/15] - Create
*)
VAR CONSTANT
	VARS_Max	: BYTE := 32;
END_VAR
VAR_INPUT
	(* Settings *)
	ID			: BYTE;
	IP			: STRING;
	PORT		: WORD:=502;
	(* Interface *)
	MB_MASTER	: ETHERNET_MODBUSMASTER_TCP;
	MB_READBUF	: ARRAY [0..128] OF WORD;
	MB_WRITEBUF : ARRAY [0..128] OF WORD;
	MB_Start	: BOOL;
	MB_Lock		: BOOL;
	(* Variables management *)
	VARS_En		: BOOL;
	VARS		: ARRAY [0..VARS_Max] OF typ_MODBUS_VAR;
	VARS_Check	: BOOL;
	VARS_Alarm	: BOOL;
	(* Variables allocation *)
	VAR_Pointer : POINTER TO ARRAY[0..99] OF WORD;
	VAR_Cfg		: POINTER TO typ_MODBUS_VAR;

	w_DO_01:BOOL;
	w_DO_02:BOOL;



END_VAR
VAR_OUTPUT
	(* Status *)
	Status_Log	: BYTE;
	Status_Vis	: DWORD;
END_VAR
VAR
	sta         : BYTE :=0;
	i			: BYTE;
	j			: BYTE;
	Alarm		: FLT_EVENT;

	VarTmr		: TON := (PT:=T#1s);
	VarSta		: BYTE; (* Status *)
	VarCnt		: BYTE; (* Scan counter *)
	VarRetry	: BYTE;
	retryErrMax	:	BYTE := 8;
	VarAlarm	: BYTE; (* Last variable with errors *)


	state : INT;
	ReadTmr		:	TON := (PT:=T#5s);
	retry		:	BYTE;
	retryErr	:	BYTE;

	ErroreComuModBus: BOOL;
	fModbusAlr:BOOL;

	MB_RegistriHoldingLetti: ARRAY [0..300] OF WORD;

	x: INT;

	(* da diego per gestione stato stringa > 255*)
	temp :STRING(255);
	tempRaw		: ARRAY [0..MAX_SEND_TCP_CLIENT] OF BYTE;
	tempRawLen :DINT;
	longString:STRING(300);

	DI_01:BOOL;
	DI_02:BOOL;
	DI_03:BOOL;
	DI_04:BOOL;
	AI_01:INT;
	AI_02:INT;
	DO_01:BOOL;
	DO_02:BOOL;


	TimeOutModBus: TON;
	ErroreTimeOut: BOOL;
	AppoggioDWORD: DWORD;


	WordLW: WORD;
	WordHI: WORD;
	ValoreDWord: DWORD;
	ValoreDint: DINT;
	testINT1: DINT;
	testINT2: DINT;
	testmoreno: BOOL;
	testmoreno1: BOOL;
END_VAR
CASE state OF
	0:	(* Refresh time manager *)
		ReadTmr(IN:=NOT ReadTmr.Q,pt:=t#1000ms);
			MB_Start:=FALSE;

		(*A tempo interrogo il nodo sempre che non ci sia qualcuno che lo sta interrogando in quel momento *)
		IF  ReadTmr.Q THEN
			state := 5;
		END_IF
	5:
(*	test_moreno:=MB_MASTER.xIS_CONNECTED;
	test_moreno1:=MB_MASTER.wERROR;
	test_moreno2:=MB_MASTER.bRESPONSE_UNIT_ID; *)
		IF  MB_MASTER.xIS_CONNECTED THEN
			state :=10;
		END_IF
	(**** Leggo le Analogiche a Disposzione  ****)

	10:	(* richiedo lettura Holding Registere   *)

			MB_MASTER.bUNIT_ID := 1;
			MB_MASTER.bFUNCTION_CODE:=3;
			MB_MASTER.wREAD_ADDRESS:=0;
			MB_MASTER.wREAD_QUANTITY:=16;
			MB_Start:=TRUE;
			state := 20;


	20:	(* Risposta all'interrogazione *)
		IF NOT MB_Start THEN
			IF MB_MASTER.wERROR<>MB_NO_ERROR THEN
				state:=300;
			ELSE

				FOR x:=0 TO MB_MASTER.wREAD_QUANTITY DO
					MB_RegistriHoldingLetti[x+MB_MASTER.wREAD_ADDRESS] := MB_READBUF[x];
				END_FOR



			DI_01:=INT_TO_BOOL (MB_RegistriHoldingLetti[11]);
			DI_02:=INT_TO_BOOL ( MB_RegistriHoldingLetti[12]);
			DI_03:=INT_TO_BOOL ( MB_RegistriHoldingLetti[13]);
			DI_04:=INT_TO_BOOL( MB_RegistriHoldingLetti[14]);
			AI_01:=WORD_TO_INT (MB_RegistriHoldingLetti[3]);
			AI_02:=WORD_TO_INT ( MB_RegistriHoldingLetti[5]);
			DO_01:=INT_TO_BOOL ( MB_RegistriHoldingLetti[8]);
			DO_02:= INT_TO_BOOL (MB_RegistriHoldingLetti[9]);

	(*		MB_MASTER.wREAD_ADDRESS:=180;
			MB_MASTER.wREAD_QUANTITY:=4;
			MB_Start:=TRUE;  *)
			state := 30;

			END_IF
		END_IF

	30:	(* Scrivo le uscite  *)



			MB_WRITEBUF[0].0:=w_DO_01 OR testmoreno1;
			MB_WRITEBUF[0].1:=w_DO_02 OR testmoreno;

			MB_MASTER.bUNIT_ID := ID;
			MB_MASTER.bFUNCTION_CODE:=6;


			MB_MASTER.wWRITE_ADDRESS:=7;
			MB_MASTER.wWRITE_QUANTITY:=1;
			MB_Start:=TRUE;
			state := 40;

	40:	(* Risposta all'interrogazione *)
		IF NOT MB_Start THEN
			IF MB_MASTER.wERROR<>MB_NO_ERROR THEN
				state:=300;
			ELSE

				state :=295;

			END_IF
		END_IF

	295:
		IF NOT MB_Start THEN
			IF  MB_MASTER.wERROR<>MB_NO_ERROR THEN (*OR ModBus.MB_MASTER.MB_Error<>0 THEN*)
				state := 300;
			ELSE
				retryErr := 0;
				retry := 0;
				state := 0;
					IF ErroreComuModBus=TRUE THEN
						LogEv(EL_Log,EO_MODBUS_TCP,ID,2,'Comunicazione_ristabilita');
						ErroreComuModBus := FALSE;
						fModbusAlr := FALSE;

				(*	WarningCtr := SEL(WarningCtr=0, WarningCtr-1, 0); *)
					END_IF
			END_IF
		END_IF



	(**** CHECK MODBUS ERROR ****)
	300: 	(* Release MODBUS *)
			retry:=retry+1;
			IF retry>3 THEN
				retry:=0;

				(* Verify if slave is dead *)
				IF retryErr < retryErrMaX THEN
					retryErr := retryErr + 1;
				ELSE
					fModbusAlr := TRUE;
					(* Verify ModBus error	*)

					IF fModbusAlr AND ErroreComuModBus=FALSE THEN
						LogEv(SEL(MB_MASTER.wERROR>0,EL_Wrn,EL_Alarm),EO_MODBUS_TCP,ID,1,WORD_TO_STRING(MB_MASTER.wERROR));
						ErroreComuModBus := TRUE;
					END_IF
				END_IF

				END_IF
			state:=0;
END_CASE



MB_MASTER( strIP_ADDRESS:=IP, wPORT:=PORT, tTIME_OUT:=T#750MS, (*xCONNECT:=TRUE,*)
		   ptREAD_DATA:=ADR(MB_READBUF), ptSEND_DATA:=ADR(MB_WRITEBUF), xSEND:=MB_Start );

IF state<>0 THEN
	MB_MASTER.xCONNECT:=TRUE;
ELSE
	MB_MASTER.xCONNECT:=FALSE;
END_IF


TimeOutModBus(In:=state<>0,PT:=t#5s);
IF TimeOutModBus.Q THEN
	State:=300;
END_IF


(* Log/visu status *)
   IF Alarm.IN   THEN Status_Log:=2; Status_Vis:=COLOR_RED;
ELSIF Vars_Alarm OR ErroreComuModBus  THEN
	Status_Log:=1; Status_Vis:=COLOR_YELLOW;
  ELSE
	Status_Log:=0; Status_Vis:=COLOR_GREEN;
END_IF
END_FUNCTION_BLOCK
ACTION VAR_Search:
(* Search VAR with specific pointer if not found return first free VAR
	[Last VAR is not active... used as safe area...] 
*)
j:=VARS_Max;
FOR i := 0 TO VARS_Max-1 DO
	IF VARS[i].Variable=0 AND j>i THEN j:=i; END_IF
	IF VARS[i].Variable=VAR_Pointer THEN
		VAR_Cfg:=ADR(VARS[i]);
		RETURN;
	END_IF
END_FOR
VAR_Cfg:=ADR(VARS[j]);
END_ACTION
ACTION VARS_Process:
(* Update var timers *)
VarTmr(IN:=(NOT VarTmr.Q));
IF VarTmr.Q THEN
	FOR i := 0 TO VARS_Max DO
		IF VARS[i].Refresh_Cnt>0 THEN VARS[i].Refresh_Cnt:=VARS[i].Refresh_Cnt-1; END_IF
	END_FOR
	VARS_Check:=TRUE;
END_IF


(* Process status *)
CASE VarSta OF
	0: (* === Init *)
		VarCnt:=0;
		VarSta:=1;

	1: (* === Wait check signal *)
		IF VARS_Check THEN
			VARS_Check:=FALSE;
			VarCnt:=0;
			VarSta:=2;
		END_IF

	2: (* === Check loop *)
		IF NOT (MB_Lock OR MB_Start) THEN
			WHILE VarCnt<=(VARS_Max-1) AND VarSta=2 DO
				(* Check only active vars *)
				IF VARS[VarCnt].Variable<>0 THEN
					(* Check var auto-refresh on timer checks *)
					IF VARS[VarCnt].Refresh_Time>0 AND VARS[VarCnt].Refresh_Cnt=0 THEN
						VARS[VarCnt].Refresh_Cnt:=VARS[VarCnt].Refresh_Time;
						VarSta:=3;
					END_IF
					(* Check refresh for change or request *)
					CASE VARS[VarCnt].FunCode OF
						5,6,15,16: (* Write functions *)
							IF VARS[VarCnt].Variable_Size=1 THEN
								IF VARS[VarCnt].Variable^<>VARS[VarCnt].Variable_Mirror THEN
									VARS[VarCnt].Variable_Mirror:=VARS[VarCnt].Variable^;
									VarSta:=3;
								END_IF
							ELSE
								IF VARS[VarCnt].Variable_Mirror<>0 THEN
									VARS[VarCnt].Variable_Mirror:=0;
									VarSta:=3;
								END_IF
							END_IF
						1,2,3,4: (* Write functions *)
							IF VARS[VarCnt].Variable_Mirror<>0 THEN
								VARS[VarCnt].Variable_Mirror:=0;
								VarSta:=3;
							END_IF
					END_CASE
				END_IF
				(* Process query *)
				IF VarSta=3 THEN
					MB_Lock:=TRUE;
					MB_MASTER.bUNIT_ID:=VARS[VarCnt].SlaveAddress;
					MB_MASTER.bFUNCTION_CODE:=VARS[VarCnt].FunCode;
					CASE VARS[VarCnt].FunCode OF
						16#5,16#6,16#F,16#10:
							MB_MASTER.wREAD_ADDRESS:=0;
							MB_MASTER.wREAD_QUANTITY:=0;
							MB_MASTER.wWRITE_ADDRESS:=VARS[VarCnt].FunAddress;
							MB_MASTER.wWRITE_QUANTITY:=VARS[VarCnt].Variable_Size;
							IF VARS[VarCnt].Variable_Size=200 THEN
								COPY_32SWAP16(VARS[VarCnt].Variable, ADR(MB_WRITEBUF));
							ELSIF VARS[VarCnt].Variable_Size>1 THEN
								MEMCPY(VARS[VarCnt].Variable, ADR(MB_WRITEBUF), 2*VARS[VarCnt].Variable_Size);
							ELSE
								MB_WRITEBUF[0]:=VARS[VarCnt].Variable^;
							END_IF
						16#1,16#2,16#3,16#4:
							MB_MASTER.wREAD_ADDRESS:=VARS[VarCnt].FunAddress;
							IF VARS[VarCnt].Variable_Size=200 THEN MB_MASTER.wREAD_QUANTITY:=2; ELSE
							  MB_MASTER.wREAD_QUANTITY:=VARS[VarCnt].Variable_Size;
							END_IF
							MB_MASTER.wWRITE_ADDRESS:=0;
							MB_MASTER.wWRITE_QUANTITY:=0;
					END_CASE
					VarRetry:=0;
					MB_Start:=TRUE;
				ELSE
					VarCnt:=VarCnt+1;
				END_IF
			END_WHILE
			(* Check loop completed -> no actions *)
			IF VarSta=2 THEN VarSta:=1; END_IF
		END_IF

	3: (* === Wait & process MB response *)
		IF NOT MB_Start THEN
			IF MB_MASTER.wERROR=0 THEN
				CASE VARS[VarCnt].FunCode OF
					1,2,3,4:
						IF VARS[VarCnt].Variable_Size=200 THEN
							COPY_32SWAP16(ADR(MB_READBUF), VARS[VarCnt].Variable);
						ELSIF VARS[VarCnt].Variable_Size>1 THEN
							MEMCPY(ADR(MB_READBUF), VARS[VarCnt].Variable, 2*VARS[VarCnt].Variable_Size);
						ELSE
							VARS[VarCnt].Variable^:=MB_READBUF[0];
						END_IF
				END_CASE
				MB_Lock:=FALSE;
				(* Signal error recovery *)
				IF VARS_Alarm=TRUE AND VarCnt=VarAlarm THEN
					LogEv(EL_Wrn,EO_MODBUS_TCP,ID,5,'');
					VARS_Alarm:=FALSE;
				END_IF
				(* Next var *)
				VarCnt:=VarCnt+1;
				VarSta:=2;
			ELSE
				IF VarRetry<10 THEN
					VarRetry:=VarRetry+1;
					MB_Start:=TRUE;
				ELSE
					MB_Lock:=FALSE;
					(* Signal error *)
					IF VARS_Alarm=FALSE THEN
						LogEv(EL_Wrn,EO_MODBUS_TCP,ID,3,WORD_TO_STRING(MB_MASTER.wERROR));
						VARS_Alarm:=TRUE;
						VarAlarm:=VarCnt-1;
					END_IF
					(* Next var *)
					VarCnt:=VarCnt+1;
					VarSta:=2;
				END_IF
			END_IF
		END_IF

ELSE
	VarSta:=0;
END_CASE
END_ACTION

(* POU Plant_Objects/obj_CRON_EDITOR_01, ST *)
FUNCTION_BLOCK obj_CRON_EDITOR_01
(* === EDITOR CRONOGRAFO ===
   v1.0[16/04/15] - Versioning
   v1.1[19/05/15] - Create empty profile when not found
*)
VAR_INPUT

	(* Common selections *)
	CN_Sel:			BYTE:=1;
	CN_Act:			BYTE;
	CN_YSel:		WORD:=2015;
	CN_YAct:		WORD;

	(* Profile editor *)
	PR_Sel: 		BYTE:=1;
	PR_Act:			BYTE;
	PR_TT:			REAL;
	PR:				typ_Cron_Profile;
	(* Profile signals *)
	PR_Load:		BOOL;
	PR_Save:		BOOL;

	(* Calendar editor *)
	CA_Sel:			BYTE:=1; (* Calendar month selected *)
	CA_Act:			BYTE;    (* Calendar month active *)
	CA_DayF:		BYTE:=0;
	CA_DayL:		BYTE:=31;
	CA_TPR:			BYTE;
	CA:				typ_Cron_Calendar; (* Only used for first 32 entries *)
	(* Calendar signals *)
	CA_Load:		BOOL;
	CA_Save:		BOOL;

	(* Jolly editor *)
	JL:				ARRAY[0..9] OF typ_Cron_Jolly;
	(* Jolly signals *)
	JL_Load:		BOOL;
	JL_Save:		BOOL;

END_VAR
VAR_OUTPUT
	Message		: STRING;
END_VAR
VAR
	sFileName	: STRING;
	sFileMode	: STRING;
	hFile		: DWORD;
	Buf			: ARRAY[0..512] OF BYTE; (* AVOID THIS!! *)

	i			: WORD;
	ver			: BYTE;
	r1			: BOOL;
	r2			: DWORD;

	x: INT;
	maxProfili: INT;

	sFileNameOld	: STRING;
	sFileModeOld		: STRING;
	hFileOld			: DWORD;




	strAppoggio: STRING;
	FileGiaCreato: BOOL;
	fileCopiato: UDINT;

	tempMultiAnnoMax:INT;
	tempMultiAnnoIndex:INT;
	TEMP_MULTIANNO_MAX_DELTA:INT:=5;
	tempRicercaFileAnno:INT;
	tempAnno:INT;
	tempTrovato:BOOL;
END_VAR
IF PR_Load THEN PR_Load_Exe();
	PR_Load:=FALSE;
END_IF
IF PR_Save THEN
PR_Save_Exe();
PR_Save:=FALSE;
END_IF
IF CA_Load THEN
CA_Load_Exe();
CA_Load:=FALSE;
END_IF
IF CA_Save THEN
CA_Save_Exe();
CA_Save:=FALSE;
END_IF
IF JL_Load THEN
JL_Load_Exe();
JL_Load:=FALSE;
END_IF
IF JL_Save THEN
 JL_Save_Exe();
 JL_Save:=FALSE;
 END_IF
END_FUNCTION_BLOCK
ACTION CA_Load_Exe:
sFileMode:='r';
FileOpen();

IF hFile<>0 THEN

	(* Read calendar month *)
	FOR i := 0 TO 31 DO
		r1:=SysFileSetPos(File:=hFile, Pos:=(1024 + ((CA_Sel-1)*32 + i)*4));
		r2:=SysFileRead(File:=hFile, Buffer:=ADR(CA.Profile[i]), Size:=1);
	END_FOR

	(* Close file *)
	SysFileClose(File:=hFile);

	(* Validate data *)
	CA_Act :=CA_Sel;
	CN_Act :=CN_Sel;
	CN_YAct:=CN_YSel;

	Message:='Calendar load OK';

END_IF
END_ACTION
ACTION CA_Save_Exe:
sFileMode:='a';
FileOpen();

IF hFile<>0 THEN

	(* Write calendar month *)
	FOR i := 0 TO 31 DO
		r1:=SysFileSetPos(File:=hFile, Pos:=(1024 + ((CA_Sel-1)*32 + i)*4));
		r2:=SysFileGetPos(hFile);
		r2:=SysFileWrite(File:=hFile, Buffer:=ADR(CA.Profile[i]), Size:=1);
	END_FOR

	(* Close file *)
	SysFileClose(File:=hFile);

	Message:='Calendar save OK';

	(* db commentato! non salva i profili, ma solo il profilo corrente, che può anche essere modificato!*)
          (*PR_Save_exe();*)
	(* nel salvare il calendario aggiorno anche i profili così ho il file completo dei profili *)


END_IF

IF hFile<>0 THEN SysFileClose(File:=hFile); END_IF (*diego add*)
END_ACTION
ACTION FileOpen:
(* Create current filename 'yyyyCRnn.DAT' *) (* creo il nome del file da aparire *)
sFileName:=CONCAT(FilesPath,WORD_TO_STRING(CN_YSel));
sFileName:=CONCAT(STR1:=sFileName, STR2:='CR');
IF CN_Sel<10 THEN
sFileName:=CONCAT(STR1:=sFileName, STR2:='0');
END_IF
sFileName:=CONCAT(STR1:=sFileName, STR2:=BYTE_TO_STRING(CN_Sel));
sFileName:=CONCAT(STR1:=sFileName, STR2:='.DAT');


(* Apro il fiel in lettura per verificare se è presente altrimenti devo crearne uno nuovo a duplicare quello dell'anno precedente - apro 1  *)
hFile:=SysFileOpen(FileName:=sFileName, Mode:='r');
FileGiaCreato:=FALSE;

tempAnno:=CN_YSel;
tempTrovato:=FALSE;

(* File non trovato da creare  *)
IF hFile=0 THEN

	 (*cerco i file precendti: dall'anno prima fino a - TEMP_MULTIANNO_MAX_DELTA*)
	 tempRicercaFileAnno:=1;

	WHILE tempRicercaFileAnno<=TEMP_MULTIANNO_MAX_DELTA AND NOT tempTrovato DO


		strAppoggio:=INT_TO_STRING(tempAnno);
		(* Verifico se esite un file da cui partire *)
		StrAppoggio:=WORD_TO_STRING(STRING_TO_WORD(strAppoggio)-tempRicercaFileAnno);
		sFileNameOld:=CONCAT(FilesPath,StrAppoggio);

		sFileNameOld:=CONCAT(STR1:=sFileNameOld, STR2:='CR');
		IF CN_Sel<10 THEN
			sFileNameOld:=CONCAT(STR1:=sFileNameOld, STR2:='0');
		END_IF
		sFileNameOld:=CONCAT(STR1:=sFileNameOld, STR2:=BYTE_TO_STRING(CN_Sel));
		sFileNameOld:=CONCAT(STR1:=sFileNameOld, STR2:='.DAT');

		(* Apro il file in lettura per la verifica della presenza del file da copiare  *)
		hFileold:=SysFileOpen(FileName:=sFileNameOld, Mode:='r');

		IF hFileold<>0 THEN

			tempTrovato:=TRUE;

			fileCopiato:=SysFileCopy(sFileName,sFileNameold);

    		   	FileGiaCreato:=fileCopiato<>0;

			IF FileGiaCreato THEN
				Message:='File Sorgente/copia  trovato - file Copiato';
			ELSE
				Message:='File Sorgente/copia  trovato - file NON Copiato';
			END_IF


			(* Chiudo il file aperto per la verifica del file presente *)
			SysFileClose(File:=hFile);
			(* Chiudo il file aperto in lettura per la verifica della presenza del file da copiare  *)
			SysFileClose(File:=hFileold);

		END_IF

		tempRicercaFileAnno:=tempRicercaFileAnno+1;

	END_WHILE

	(* se non ho trovato nessun file..lo creo vuoto*)
	IF tempTrovato=FALSE THEN   (* file non trovato quindi devo crearne uno nuovo *)

			(* Create empty file *)
			hFile:=SysFileOpen(FileName:=sFileName, Mode:='w');
			MEMCLR(pDestinationAddress:=ADR(Buf), BytesToClear:=SIZEOF(Buf));
			FOR i := 0 TO 10239 BY 512 DO
				SysFileWrite(File:=hFile, Buffer:=ADR(Buf), Size:=512);
			END_FOR

			Buf[0]:=1;
			SysFileSetPos(File:=hFile, Pos:=0);
			SysFileWrite(File:=hFile, Buffer:=ADR(Buf), Size:=1);

			(* Chiudo il file aperto per la verifica del file presente *)
			SysFileClose(File:=hFile);
			(* Chiudo il file aperto in lettura per la verifica della presenza del file da copiare  *)
			SysFileClose(File:=hFileold);

			Message:='File Sorgente/copia non trovato-file Vuoto';

	END_IF


ELSE

	(* Chiudo il file aperto per la verifica del file presente *)
	SysFileClose(File:=hFile);

END_IF




(* Apro il file per permettere la scrittura o la lettura del file da parte delle altre action . la chiusura del file è delegata alle Action *)
hFile:=SysFileOpen(FileName:=sFileName, Mode:=sFileMode);
END_ACTION
ACTION JL_Load_Exe:
sFileMode:='r';
FileOpen();

IF hFile<>0 THEN

	(* Read jolly *)
	r1:=SysFileSetPos(File:=hFile, Pos:=512);
	r2:=SysFileRead(File:=hFile, Buffer:=ADR(JL), Size:=SIZEOF(JL));

	(* Close file *)
	SysFileClose(File:=hFile);

	(* Validate data *)
	CN_Act:=CN_Sel;
	CN_YAct:=CN_YSel;

	Message:='Jolly load OK';

END_IF
END_ACTION
ACTION JL_Save_Exe:
sFileMode:='a';
FileOpen();

IF hFile<>0 THEN

	(* Write selected profile *)
	r1:=SysFileSetPos(File:=hFile, Pos:=512);
	r2:=SysFileWrite(File:=hFile, Buffer:=ADR(JL), Size:=SIZEOF(JL));

	(* Close file *)
	SysFileClose(File:=hFile);

	Message:='Jolly save OK';

END_IF
END_ACTION
ACTION PR_Load_Exe:
sFileMode:='r';
FileOpen();

IF hFile<>0 THEN

	(* Read selected profile *)
	r1:=SysFileSetPos(File:=hFile, Pos:=(3072 + 512*PR_Sel));
	r2:=SysFileRead(File:=hFile, Buffer:=ADR(PR), Size:=SIZEOF(PR));

	(* Close file *)
	SysFileClose(File:=hFile);

	(* Validate data *)
	PR_Act:=PR_Sel;
	CN_Act:=CN_Sel;
	CN_YAct:=CN_YSel;

	Message:='Profile load OK';

END_IF
END_ACTION
ACTION PR_Save_Exe:
sFileMode:='a';
FileOpen();

IF hFile<>0 THEN

		(* Write selected profile *)
		r1:=SysFileSetPos(File:=hFile, Pos:=(3072 + 512*PR_Sel));
		r2:=SysFileWrite(File:=hFile, Buffer:=ADR(PR), Size:=SIZEOF(PR));

		(* Close file *)
		SysFileClose(File:=hFile);

		Message:='Profile save OK';

END_IF

IF hFile<>0 THEN SysFileClose(File:=hFile); END_IF (*diego add*)
END_ACTION
ACTION PR_Save_Exe_Multi:
(*eseguo  salvataggio profilo per l'anno corrente del CronoEditor - quello indicato da CN_YSel*)
CronEd.PR_Save_Exe();

(*verifico se esistono i file di schedulazioni per anni successivi: se aggiorno i profili anche lì*)

(*tempMultiAnnoMax dice fino a quale anno si considera*)
tempMultiAnnoMax:=CronEd.CN_YSel+TEMP_MULTIANNO_MAX_DELTA;

(* per ogni anno, vrifico se esiste il relativo file e se si aggiorno i profili anche li *)
FOR tempMultiAnnoIndex:=CronEd.CN_YSel+1 TO tempMultiAnnoMax BY 1 DO

	sFileName:=CONCAT(FilesPath,INT_TO_STRING(tempMultiAnnoIndex));
	sFileName:=CONCAT(STR1:=sFileName, STR2:='CR');
	IF CN_Sel<10 THEN
		sFileName:=CONCAT(STR1:=sFileName, STR2:='0');
	END_IF
	sFileName:=CONCAT(STR1:=sFileName, STR2:=INT_TO_STRING(CN_Sel));
	sFileName:=CONCAT(STR1:=sFileName, STR2:='.DAT');

	hFile:=SysFileOpen(FileName:=sFileName, Mode:='r');
	(* file esiste, aggiorno profili per quell'anno *)
	IF hFile<>0 THEN

		SysFileClose(File:=hFile);
		CronEd.CN_YSel:=tempMultiAnnoIndex;
		CronEd.PR_Save_Exe();

	ELSE
		SysFileClose(File:=hFile);

	END_IF


END_FOR
END_ACTION

(* POU Plant_Objects/obj_CRONTER_01, ST *)
FUNCTION_BLOCK obj_CRONTER_01
(* === THERMOSTAT ===
   v1.0[30/07/15] - Versioning
*)
VAR_INPUT
	(* Settings *)
	ID			: BYTE;		(* Index of instanced object *)

	InitOK		: BOOL;
	Alarm		: BOOL;
	Warning		: BOOL;

	Profile		: typ_Cron_Profile; 				(* Profilo attivo *)
	ProfileNr	: BYTE;								(* Indice profilo attivo *)
	CalendarIdx : WORD;								(* Indice calendario attivo *)
	Jolly		: ARRAY[0..9] OF typ_Cron_Jolly;	(* Jolly attivi *)

	Temperature	: INT;
	Local_MaxRunTAmb	:	INT;					(* Local maximum environment temperature, NOT "TAMB" *)
	Histeresys:INT; (* isteresi per la ripartenza del Comando ON*)


	sFile: 	STRING;


END_VAR
VAR_IN_OUT
END_VAR
VAR_OUTPUT
	SetPoint		: INT;
	Run				: BOOL;
	AntifreezeForce	: BOOL;
	RunCrono		: BOOL;

	(* Status *)
	Status_Log		: BYTE;
	Status_Vis 		: DWORD;
END_VAR
VAR
	Buf: 	ARRAY[0..512] OF BYTE; (* AVOID THIS!! *)
	hFile: 	DWORD;

	sFile2: STRING;

	i:		WORD;
	t1:		DWORD;
	t2:		BOOL;

END_VAR
(* Check initialization *)
(*IF NOT InitOK THEN Init(); END_IF*)

(* Check Temperature *)
IF Temperature <Local_MaxRunTAmb THEN

	(* LOCAL environment temperature lower than maximum allowed -> Proceed with SetPoint adjustment *)
	(* Chrono *)
(*	IF CalendarIdx<>Sys.Time_CT_Day THEN DB_Load(); END_IF *)

	IF CalendarIdx<>Sys.Time_CT_Day OR InitOK=FALSE THEN  (* col cambio della data carico il file corretti dove è intergrato il controllo della presenza del file *)
		CronEd(CN_Sel:=WORD_TO_BYTE(id),CN_YSel:=Sys.Time_Year, CA_Load:=TRUE,PR_Load:=TRUE);
		DB_Load(	sFile:= CronEd.sFileName);  (* aggiorno il SetPoint  partendo dal file noto*)
		InitOK:=TRUE;
	END_IF


	SetPoint:=Profile.Setpoint[Sys.Time_CT_Quarter];

	(* Check jolly *)
	FOR i := 0 TO 9 DO
		IF ( DT_TO_DWORD(Jolly[i].Start)>0  AND Jolly[i].End>Jolly[i].Start AND
		     Jolly[i].Start<=Sys.Time_CT_DT AND Jolly[i].End>Sys.Time_CT_DT ) THEN
				SetPoint:=Jolly[i].Temp;
		END_IF
	END_FOR

(*
	IF SetPoint < 180 THEN
		(* Switch off the device *)
		Run := FALSE;
	ELSE
		(* Set according to feedback T - Histeresys of 1°C *)
		IF Temperature >= (SetPoint + 5) THEN
			Run := FALSE;
		ELSIF Temperature <= (SetPoint - 5) THEN
			Run := TRUE;
		END_IF

		(* Between "SetPoint-5" and "SetPoint+5" last state (ON or OFF) of "Run" is kept	*)
	END_IF
*)
(* Gestione uscita Crono *)
		IF SetPoint>0 THEN RunCrono := TRUE;
		ELSIF SetPoint=0 THEN RunCrono := FALSE;
		END_IF

(* GEstione uscita Cronotermostato *)

		IF Temperature >= (SetPoint) THEN
			Run := FALSE;
		ELSIF Temperature <= (SetPoint - Histeresys) THEN
			Run := TRUE;
		END_IF
ELSE
	(* Environment overtemperature: stop heating -> Stop device *)
	Run := FALSE;
END_IF

(* Freeze warning: Switch on and heat! *)
(*IF Temperature < Plant_AntiFreezeTAmb THEN AntifreezeForce := TRUE;
ELSE AntifreezeForce := FALSE;
END_IF*)



(* Status color *)
   IF Alarm   THEN Status_Log:=2; Status_Vis:=COLOR_RED;
ELSIF Warning THEN Status_Log:=1; Status_Vis:=COLOR_YELLOW;
              ELSE Status_Log:=0; Status_Vis:=COLOR_GREEN;
			  END_IF
END_FUNCTION_BLOCK
ACTION AddLogData:
Logger.s1:=INSERT('&THER=',BYTE_TO_STRING(ID),5);
IF ID<10 THEN Logger.s1:=INSERT(Logger.s1,'0',5); END_IF

Logger.s1:=CONCAT(Logger.s1,INT_TO_STRING(SetPoint));			Logger.s1:=CONCAT(Logger.s1,';');

Logger.s1:=CONCAT(Logger.s1,WORD_TO_STRING(Status_Log));
ADDSTRING(ADR(Logger.TData), ADR(Logger.s1), Logger.TLen);
END_ACTION
ACTION DB_Create:
(* Create empty file *)
hFile:=SysFileOpen(FileName:=sFile, Mode:='w');

MEMCLR(pDestinationAddress:=ADR(Buf), BytesToClear:=SIZEOF(Buf));
FOR i := 0 TO 10239 BY 512 DO
	t1:=SysFileWrite(File:=hFile, Buffer:=ADR(Buf), Size:=512);		(* Clear created file (all bytes 0) *)
END_FOR
Buf[0]:=1;
t2:=SysFileSetPos(File:=hFile, Pos:=0);
t1:=SysFileWrite(File:=hFile, Buffer:=ADR(Buf), Size:=1);
SysFileClose(File:=hFile);
END_ACTION
ACTION DB_Load:
(*

DB_SetName();


(* File not found *)
IF hFile=0 THEN
	Warning:=TRUE;
	LogEv(EL_Wrn,EO_CRON,ID,1,'No_data_file');
	DB_Create();
	(* Reopen file *)
	hFile:=SysFileOpen(FileName:=sFile, Mode:='r');
	IF hfile=0 THEN
		Alarm:=TRUE;
		LogEv(EL_Alarm,EO_CRON,ID,3,'Filesystem_error');
		RETURN;
	END_IF
END_IF
*)

(* Open data file *)
hFile:=SysFileOpen(FileName:=sFile, Mode:='r');

(* Check version *)
SysFileRead(File:=hFile, Buffer:=ADR(Buf), Size:=1);
IF Buf[0]<>1 THEN
	IF NOT Alarm THEN
		Alarm:=TRUE;
		LogEv(EL_Alarm,EO_CRON,ID,2,'Bad_data_version');
	END_IF
	SysFileClose(File:=hFile);
	RETURN;
END_IF

(* Read Jolly data *)
t2:=SysFileSetPos(File:=hFile, Pos:=512);
t1:=SysFileRead(File:=hFile, Buffer:=ADR(Jolly), Size:=SIZEOF(Jolly));
(* Read active profile index *)
CalendarIdx:=Sys.Time_CT_Day;
t2:=SysFileSetPos(File:=hFile, Pos:=(1024+4*CalendarIdx));
t1:=SysFileRead(File:=hFile, Buffer:=ADR(ProfileNr), Size:=SIZEOF(ProfileNr));
(* Read active profile *)
t2:=SysFileSetPos(File:=hFile, Pos:=(3072+512*ProfileNr));
t1:=SysFileRead(File:=hFile, Buffer:=ADR(Profile), Size:=SIZEOF(Profile));

(* Close file and validate data *)
SysFileClose(File:=hFile);
END_ACTION
ACTION DB_SetName:
(* Create current filename 'yyyyCRnn.DAT' *)
sFile:=CONCAT(FilesPath,WORD_TO_STRING(Sys.Time_Year));
sFile:=CONCAT(STR1:=sFile, STR2:='CR');
IF ID<10 THEN
sFile:=CONCAT(STR1:=sFile, STR2:='0');
END_IF
sFile:=CONCAT(STR1:=sFile, STR2:=BYTE_TO_STRING(ID));
sFile:=CONCAT(STR1:=sFile, STR2:='.DAT');
END_ACTION
ACTION Init:
DB_Load();
InitOK:=TRUE;
END_ACTION

(* POU Plant_Objects/obj_LuxSimple, ST *)
FUNCTION_BLOCK obj_LuxSimple
VAR
	ModeToServer : BYTE;
	ForcedOn : BYTE;
	ForcedOff : BYTE;

(* controllo errori *)
	sLux_EN			: FLT_EVENT;
	chkLux_ST		: FLT_TIME := ( TTAP:=T#20S, INITEV:=FALSE );


(* controllo energia *)
	TickTimer		: TON := ( PT:=T#1S );



END_VAR
VAR_INPUT
	ID					: WORD;
	DimmingType		: BYTE := 0;	 (* /0: no dimming (digital), 1: dimming (analog) *)
	DimmingValForTimer	: INT := 0;	 (* /valore 0...100 del dimming di default del lux sotto timer *)

	(* Physical inputs *)
	DI_ONLux:BOOL;
	Lux_State		: BOOL; (* Status feedback *)

	(* Controls *)
	CTRL_MODE			: BYTE;	 (* 0:MAN OFF, 1:MAN-ON, 3:Timer laser, 2:Cronografo*)
	CTRL_MODE_BackUp	: BYTE:=2;	 (*Salvo il valore di default per il ripristino *)




END_VAR

VAR_IN_OUT
	WORKINGTIME		: DWORD; (* [sec] Internal working time counter *)
	POWERONCYCLES		: WORD;	(* DWORD; Internal counter of power-on cycles *)
	ENERGYCOUNTER		: WORD;	(* DWORD;  [E-1 kWh] Internal energy counter *)
	ENERGYCOUNTER_t 	: DWORD; (* Temporary energy in E-2*Wsec *)
END_VAR



VAR_OUTPUT
	(* uscite fisiche *)
	Lux_Enable : BOOL;
	(* Status *)
	Status_Log		: BYTE;
	Status_Vis 		: DWORD;
END_VAR
(* Controllo Accensione *)

CASE CTRL_MODE OF    (* 0:MAN OFF, 1:MAN-ON, 3:Timer laser, 2:Cronografo*)

		0: Lux_Enable:=FALSE;

		1: Lux_Enable:=TRUE;

		2: Lux_Enable:=DI_ONLux;

		3: Lux_Enable:=DI_ONLux;


END_CASE;

(* Temporary energy counter *)
TickTimer(IN:=NOT TickTimer.Q);
IF TickTimer.Q AND Lux_Enable THEN
	WORKINGTIME:=WORKINGTIME+1;
	IF ENERGYCOUNTER_t>36000000 THEN
		ENERGYCOUNTER_t:=ENERGYCOUNTER_t-36000000;
		ENERGYCOUNTER:=ENERGYCOUNTER+1;
	END_IF
END_IF


CheckFault();
END_FUNCTION_BLOCK
ACTION AddLogData:
Logger.s1:=INSERT('&LUX=',WORD_TO_STRING(ID),4);
IF ID<10 THEN Logger.s1:=INSERT(Logger.s1,'0',4); END_IF

(*Logger.s1:=CONCAT(Logger.s1,WORD_TO_STRING(REL_V));				Logger.s1:=CONCAT(Logger.s1,';');
//Logger.s1:=CONCAT(Logger.s1,WORD_TO_STRING(REL_A));				Logger.s1:=CONCAT(Logger.s1,';');
//Logger.s1:=CONCAT(Logger.s1,DWORD_TO_STRING(ENERGYCOUNTER));	Logger.s1:=CONCAT(Logger.s1,';');*)


Logger.s1:=CONCAT(Logger.s1,SEL(Lux_Enable,'0','100'));				Logger.s1:=CONCAT(Logger.s1,';');
Logger.s1:=CONCAT(Logger.s1,DWORD_TO_STRING(WorkingTime));		Logger.s1:=CONCAT(Logger.s1,';');
Logger.s1:=CONCAT(Logger.s1,DWORD_TO_STRING(PowerOnCycles));	Logger.s1:=CONCAT(Logger.s1,';');
(*//Logger.s1:=CONCAT(Logger.s1,INT_TO_STRING(REL_TEMP));			Logger.s1:=CONCAT(Logger.s1,';');*)

CASE CTRL_MODE OF
	0: 	(* Manuale OFF *)
		ModeToServer := 0;
		ForcedOn := 0;
		ForcedOff := 1;
	1:	(* Manuale ON *)
		ModeToServer := 0;
		ForcedOn := 1;
		ForcedOff := 0;	
	2:	(* Cronografo *)
		ModeToServer := 2;
		ForcedOn := 0;
		ForcedOff := 0;
	3: 	(* Timer *)
		ModeToServer := 1;
		ForcedOn := 0;
		ForcedOff := 0;
END_CASE

Logger.s1:=CONCAT(Logger.s1,BYTE_TO_STRING(ModeToServer));			Logger.s1:=CONCAT(Logger.s1,';');
Logger.s1:=CONCAT(Logger.s1,BYTE_TO_STRING(Status_Log));			Logger.s1:=CONCAT(Logger.s1,';');
Logger.s1:=CONCAT(Logger.s1,BYTE_TO_STRING(ForcedOn));			Logger.s1:=CONCAT(Logger.s1,';');
Logger.s1:=CONCAT(Logger.s1,BYTE_TO_STRING(ForcedOff));
ADDSTRING(ADR(Logger.TData), ADR(Logger.s1), Logger.TLen);
END_ACTION
ACTION CheckFault:
(* Generate status events *)
sLux_EN(IN:=Lux_Enable);
IF sLux_EN.EVL THEN
	LogEv(EL_Log,EO_LUX,ID,2,'Light_OFF'); (* Light OFF  *);
END_IF
IF sLux_EN.EVH THEN
	LogEv(EL_Log,EO_LUX,ID,3,'Light_ON'); (* Light ON  *);
	POWERONCYCLES:=POWERONCYCLES+1;
END_IF

(* Check status feedback *)
chkLux_ST(IN:=(Lux_State<>Lux_Enable));
IF chkLux_ST.EVH THEN
	LogEv(EL_Alarm,EO_LUX,ID,9,'Fail'); (*  Feedback failure - Lux_State<>Lux_Enable  *);
END_IF
IF chkLux_ST.EVL THEN
	LogEv(EL_Log,EO_LUX,ID,1,'Successful'); (*  Light feedback OK - Lux_State = Lux_Enable  *);
END_IF


(* Status color *)
IF chkLux_ST.OUT THEN
	Status_Log:=2; Status_Vis:=COLOR_RED;
ELSE
	Status_Log:=0;
	Status_Vis:=SEL(Lux_Enable,COLOR_GREEN_OFF,COLOR_GREEN);
END_IF
END_ACTION

(* POU obj_MODBUS_Free, ST *)
FUNCTION_BLOCK obj_MODBUS_Free
(* === MODBUS PROTOCOL INTERFACE ===
   v1.1[19/06/15] - Added new VARS allocation and searching
*)
VAR CONSTANT
	VARS_Max	: BYTE := 32;
END_VAR
VAR_INPUT
	(* Settings *)
	ID			: BYTE;
	COM			: BYTE;
	BAUDRATE	: COM_BAUDRATE;
	ASCIIMODE: BOOL;

	RS485		: BOOL := FALSE;


	N_STOPBits	:BYTE:=1;

 	(* Interface *)
	MB_MASTER	: MODBUS_EXTENDED_MASTER;
	MB_Start	: BOOL;
	MB_Query	: typModbusExtendedQuery;
	MB_Resp		: typModbusResponse;
	MB_Lock		: BOOL;
	MB_timeOut	: TIME := t#500ms;

	(* Variables management *)
	VARS_En		: BOOL;
	VARS		: ARRAY [0..VARS_Max] OF typ_MODBUS_VAR;
	VARS_Check	: BOOL;
	VARS_Alarm	: BOOL;

	(* Variables allocation *)
	VAR_Pointer : POINTER TO ARRAY[0..99] OF WORD;
	VAR_Cfg		: POINTER TO typ_MODBUS_VAR;
END_VAR
VAR_OUTPUT
	(* Status *)
	Status_Log	: BYTE;
	Status_Vis	: DWORD;
END_VAR
VAR
	sta         : BYTE :=0;
	i			: BYTE;
	j			: BYTE;
	Alarm		: FLT_EVENT;
	
	VarTmr		: TON := (PT:=T#1s);
	VarSta		: BYTE; (* Status *)
	VarCnt		: BYTE; (* Scan counter *)
	VarRetry	: BYTE;
	VarAlarm	: BYTE; (* Last variable with errors *)
END_VAR
IF N_STOPBits=1 THEN MB_MASTER.csCOM_STOPBITS:=STOPBITS_1;END_IF
IF N_STOPBits=2 THEN MB_MASTER.csCOM_STOPBITS:=STOPBITS_2;END_IF

MB_MASTER(ENABLE:=TRUE,	ASCII_Mode:=ASCIIMODE, bCOM_PORT:=COM, cbCOM_BAUDRATE:=BAUDRATE,
		cfCOM_FLOW_CONTROL:=SEL(RS485,NO_FLOW_CONTROL,HALFDUPLEX),
		tTIME_OUT:=MB_timeOut,	StartFunction:=MB_Start, ExtQuery:=MB_Query, Response:=MB_Resp);

(* Process variable management *)
IF VARS_En THEN VARS_Process(); END_IF

(* Check status *)
Alarm(IN:=(MB_MASTER.bInterfaceError<>0));
IF Alarm.EVH THEN
	LogEv(SEL(MB_MASTER.bInterfaceError<>3,EL_Wrn,EL_Alarm),EO_MODBUS,ID,1,BYTE_TO_STRING(MB_MASTER.bInterfaceError));
END_IF
IF Alarm.EVL THEN								(* Trigger a fall edge: MODBUS back working *)
	LogEv(EL_Log,EO_MODBUS,ID,2,'MODBUS_OK');
END_IF

(* Log/visu status *)
   IF Alarm.IN   THEN Status_Log:=2; Status_Vis:=COLOR_RED;
ELSIF Vars_Alarm THEN Status_Log:=1; Status_Vis:=COLOR_YELLOW;
  				 ELSE Status_Log:=0; Status_Vis:=COLOR_GREEN;
END_IF
END_FUNCTION_BLOCK
ACTION VAR_Search:
(* Search VAR with specific pointer if not found return first free VAR
	[Last VAR is not active... used as safe area...] 
*)
j:=VARS_Max;
FOR i := 0 TO VARS_Max-1 DO
	IF VARS[i].Variable=0 AND j>i THEN j:=i; END_IF
	IF VARS[i].Variable=VAR_Pointer THEN
		VAR_Cfg:=ADR(VARS[i]);
		RETURN;
	END_IF
END_FOR
VAR_Cfg:=ADR(VARS[j]);
END_ACTION
ACTION VARS_Process:
(* Update var timers *)
VarTmr(IN:=(NOT VarTmr.Q));
IF VarTmr.Q THEN
	FOR i := 0 TO VARS_Max DO
		IF VARS[i].Refresh_Cnt>0 THEN VARS[i].Refresh_Cnt:=VARS[i].Refresh_Cnt-1; END_IF
	END_FOR
	VARS_Check:=TRUE;
END_IF


(* Process status *)
CASE VarSta OF
	0: (* === Init *)
		VarCnt:=0;
		VarSta:=1;

	1: (* === Wait check signal *)
		IF VARS_Check THEN				(* Decremented "Refresh_Cnt" *)
			VARS_Check:=FALSE;
			VarCnt:=0;
			VarSta:=2;
		END_IF

	2: (* === Check loop *)
		IF NOT (MB_Lock OR MB_Start) THEN
			WHILE VarCnt<=(VARS_Max-1) AND VarSta=2 DO
				(* Check only active vars *)
				IF VARS[VarCnt].Variable<>0 THEN			(* "Variable" is a pointer to word, so if 0 no address *)
					(* Check var auto-refresh on timer checks *)
					IF VARS[VarCnt].Refresh_Time>0 AND VARS[VarCnt].Refresh_Cnt=0 THEN
						VARS[VarCnt].Refresh_Cnt:=VARS[VarCnt].Refresh_Time;
						VarSta:=3;
					END_IF
					(* Check refresh for change or request *)
					CASE VARS[VarCnt].FunCode OF
						5,6,15,16: (* Write functions *)
							IF VARS[VarCnt].Variable_Size=1 THEN
								IF VARS[VarCnt].Variable^<>VARS[VarCnt].Variable_Mirror THEN
									VARS[VarCnt].Variable_Mirror:=VARS[VarCnt].Variable^;
									VarSta:=3;
								END_IF
							ELSE
								IF VARS[VarCnt].Variable_Mirror<>0 THEN
									VARS[VarCnt].Variable_Mirror:=0;
									VarSta:=3;
								END_IF
							END_IF
						1,2,3,4: (* Read functions *)
							IF VARS[VarCnt].Variable_Mirror<>0 THEN
								VARS[VarCnt].Variable_Mirror:=0;
								VarSta:=3;
							END_IF
					END_CASE
				END_IF
				(* Process query *)
				IF VarSta=3 THEN
					MB_Lock:=TRUE;
					MB_Query.SlaveAddress:=VARS[VarCnt].SlaveAddress;
					MB_Query.FunctionCode:=VARS[VarCnt].FunCode;
					CASE VARS[VarCnt].FunCode OF
						16#5,16#6,16#F,16#10:
							MB_Query.Read_Quantity:=0;
							MB_Query.Read_StartAddress:=0;
							MB_Query.Write_StartAddress:=VARS[VarCnt].FunAddress;
							MB_Query.Write_Quantity:=VARS[VarCnt].Variable_Size;
							IF VARS[VarCnt].Variable_Size=200 THEN
								COPY_32SWAP16(VARS[VarCnt].Variable, ADR(MB_Query.Write_Data[0]));
							ELSIF VARS[VarCnt].Variable_Size>1 THEN
								MEMCPY(VARS[VarCnt].Variable, ADR(MB_Query.Write_Data[0]), 2*VARS[VarCnt].Variable_Size);
							ELSE
								MB_Query.Write_Data[0]:=VARS[VarCnt].Variable^;
							END_IF
						16#1,16#2,16#3,16#4:
							MB_Query.Read_StartAddress:=VARS[VarCnt].FunAddress;
							IF VARS[VarCnt].Variable_Size=200 THEN MB_Query.Read_Quantity:=2; ELSE
							  MB_Query.Read_Quantity:=VARS[VarCnt].Variable_Size;
							END_IF
							MB_Query.Write_StartAddress:=0;
							MB_Query.Write_Quantity:=0;
					END_CASE
					VarRetry:=0;
					MB_Start:=TRUE;
				ELSE
					VarCnt:=VarCnt+1;
				END_IF
			END_WHILE
			(* Check loop completed -> no actions *)
			IF VarSta=2 THEN VarSta:=1; END_IF
		END_IF

	3: (* === Wait & process MB response *)
		IF NOT MB_Start THEN
			IF MB_MASTER.MB_Error=0 THEN
				CASE VARS[VarCnt].FunCode OF
					1,2,3,4:
						IF VARS[VarCnt].Variable_Size=200 THEN
							COPY_32SWAP16(ADR(MB_Resp.Data), VARS[VarCnt].Variable);
						ELSIF VARS[VarCnt].Variable_Size>1 THEN
							MEMCPY(ADR(MB_Resp.Data), VARS[VarCnt].Variable, 2*VARS[VarCnt].Variable_Size);
						ELSE
							VARS[VarCnt].Variable^:=MB_Resp.Data[0];
						END_IF
				END_CASE
				MB_Lock:=FALSE;
				(* Signal error recovery *)
				IF VARS_Alarm=TRUE AND VarCnt=VarAlarm THEN
					LogEv(EL_Wrn,EO_MODBUS,ID,5,'');
					VARS_Alarm:=FALSE;
				END_IF
				(* Next var *)
				VarCnt:=VarCnt+1;
				VarSta:=2;
			ELSE
				IF VarRetry<3 THEN
					VarRetry:=VarRetry+1;
					MB_Start:=TRUE;
				ELSE
					MB_Lock:=FALSE;
					(* Signal error *)
					IF VARS_Alarm=FALSE THEN
						LogEv(EL_Wrn,EO_MODBUS,ID,3,INT_TO_STRING(MB_MASTER.MB_Error));
						VARS_Alarm:=TRUE;
						VarAlarm:=VarCnt-1;
					END_IF
					(* Next var *)
					VarCnt:=VarCnt+1;
					VarSta:=2;
				END_IF
			END_IF
		END_IF

ELSE
	VarSta:=0;
END_CASE
END_ACTION

(* POU Utils Functions/PLANT_STATUS, ST *)
FUNCTION_BLOCK PLANT_STATUS
VAR_INPUT
	obj_Status		:	WORD;
END_VAR
VAR_OUTPUT
END_VAR
VAR
	PLANT_STATUS	:	WORD;

	Pwm				:	TON := (PT:=T#1s);
END_VAR
CASE plant_Status OF

	0:	(* Plant OK - Everything works well *)
		Pwm(IN:=FALSE);							(* Stop timer if running *)
		LAMP_AL := FALSE;						(* Keep the lamp switched off *)

	1:	(* Plant in warning *)
		Pwm(IN:= NOT(Pwm.Q));

		IF Pwm.Q THEN
			LAMP_AL := NOT LAMP_AL;				(* Toggle output *)
		END_IF

	2:	(* Plant in alarm *)
		Pwm(IN:=FALSE);							(* Stop timer if running *)
		LAMP_AL	:= TRUE;						(* Keep the lamp switched on *)

END_CASE

plant_Status := 0;		(* Reset plant status *)
END_FUNCTION_BLOCK
ACTION UpdateStatus:
IF plant_Status = 2 THEN

	RETURN;					(* If plant already in alarm condition do nothing *)

ELSE

		IF obj_Status <> 0 THEN
			plant_Status := obj_Status;			(* If plant in warning/normal condition and current object in alarm, update plant status *)
		END_IF
END_IF
END_ACTION

(* POU PLC_WDT, ST *)
FUNCTION PLC_WDT: DWORD VAR_INPUT dwEvent: DWORD; dwFilter: DWORD; dwOwner: DWORD; END_VAR
LogEv(EL_AlarmStop,EO_SYS,1,10,'Watchdog');
END_FUNCTION

(* POU String/pSTRCAT, ST *)
(* STRCAT := STRCAT(STR1,STR2); *)
FUNCTION pSTRCAT : STRING(500)
VAR_INPUT
	STR1:	STRING(500);
	STR2:	STRING(32);
END_VAR
VAR
	ps1: POINTER TO BYTE;
	ps2: POINTER TO BYTE;
	pf:	 POINTER TO BYTE;

	ii: WORD;

END_VAR

(* versione sostitutiva thread safe della funzione CONCAT *)
(* questa funzione nasce dall'esigenza di non usare la funzione di sistema STRCAT perchè non è task safe *)

ps1 := ADR(STR1);
ps2 := ADR(STR2);

pf	:= ADR(pSTRCAT);

ii := 0;
WHILE ps1^<>0 DO
	pf^ := ps1^;
	pf := pf + 1;
	ps1:= ps1 + 1;
	ii := ii + 1;
	IF ii> 1000 THEN
		EXIT; (* termina ciclo se dimensione stringa 1 eccede per qualche motivo *)
	END_IF;

END_WHILE


WHILE ps2^<>0 DO
	pf^ := ps2^;
	pf := pf + 1;
	ps2:= ps2 + 1;
	ii := ii + 1;
	IF ii> 1000 THEN
		EXIT; (* termina ciclo se dimensione stringa 1 eccede per qualche motivo *)
	END_IF;
END_WHILE

pf^ := 0; (* termino stringa *)
END_FUNCTION

(* POU RAWTOHEXSTR, ST *)
FUNCTION RAWTOHEXSTR : STRING(128)
VAR_INPUT
	pData: POINTER TO BYTE;
	DataLen: BYTE;
END_VAR
VAR
	pt: POINTER TO BYTE;
	xl: BYTE;
END_VAR
pt:=ADR(RAWTOHEXSTR);

xl:=2;

WHILE DataLen>0 AND xl<128 DO

	pt^ := (pData^ / 16#10) + 48 + (((pData^ / 16#10)/10)*7);
	pt:=pt+1;
	pt^ := (pData^ AND 16#0F)  + 48 + (((pData^ AND 16#0F)/10)*7);
	pt:=pt+1;

	xl:=xl+2;

	DataLen:=DataLen-1;
	pData:=pData+1;

END_WHILE

pt^:=0;
END_FUNCTION

(* POU Utils/RTC_Update, ST *)
FUNCTION RTC_Update : BOOL
VAR
	T: DT;
	TS: STRING;
	TS2: STRING;
	Hour: BYTE;
	Minute: BYTE;
END_VAR
(* Get RTC time *)
T:=SysRtcGetTime(TRUE);
Sys.Time_CT_DT:=T;
(* Calculate variables *)
TS:=DT_TO_STRING(T);
Sys.Time_LogString:=DELETE(STR:=TS, LEN:=3, POS:=1);
TS2:=MID(STR:=TS, LEN:=4, POS:= 4); Sys.Time_Year 	:=STRING_TO_WORD(TS2);
TS2:=MID(STR:=TS, LEN:=2, POS:= 9); Sys.Time_Month	:=STRING_TO_BYTE(TS2);
TS2:=MID(STR:=TS, LEN:=2, POS:=12); Sys.Time_Day  	:=STRING_TO_BYTE(TS2);
Sys.Time_CT_Day:=(32*(Sys.Time_Month-1)+Sys.Time_Day-1);
TS2:=MID(STR:=TS, LEN:=2, POS:=15); Hour			:=STRING_TO_BYTE(TS2);
TS2:=MID(STR:=TS, LEN:=2, POS:=18); Minute		 	:=STRING_TO_BYTE(TS2);
Sys.Time_CT_Quarter:=Hour*4+(Minute/15);
END_FUNCTION

(* POU Utils Functions/SHIFT_ARRAY, ST *)
FUNCTION SHIFT_ARRAY : BOOL
VAR_INPUT
	pData	:	POINTER TO ARRAY [1..2] OF WORD;
	Size	:	BYTE;
END_VAR
VAR
	pNew	:	POINTER TO WORD;
	i		:	BYTE;
END_VAR
(* Shift right *)
FOR i:=1 TO (Size-1) BY 1 DO

	(*pNew := pData + 1;*)
	pData^[i] := pData^[i+1];
	(*pData := pData + 1;*)

END_FOR
END_FUNCTION

(* POU Utils Functions/TONOF, ST *)
FUNCTION_BLOCK TONOF
VAR_INPUT
	IN		: BOOL;
	PT_ON	: TIME; (* time to pass, before OUT is set *)
	PT_OF	: TIME; (* time to pass, before OUT is reset *)
END_VAR
VAR_OUTPUT
	OUT		: BOOL;
END_VAR
VAR
	timer	: TON;
END_VAR
IF IN<>OUT THEN
	timer(IN:=TRUE,PT:=SEL(IN,PT_OF,PT_ON));
	IF timer.Q THEN OUT:=IN; END_IF
ELSE
	timer(IN:=FALSE);
END_IF
END_FUNCTION_BLOCK

(* Visualisation PLC_VISU
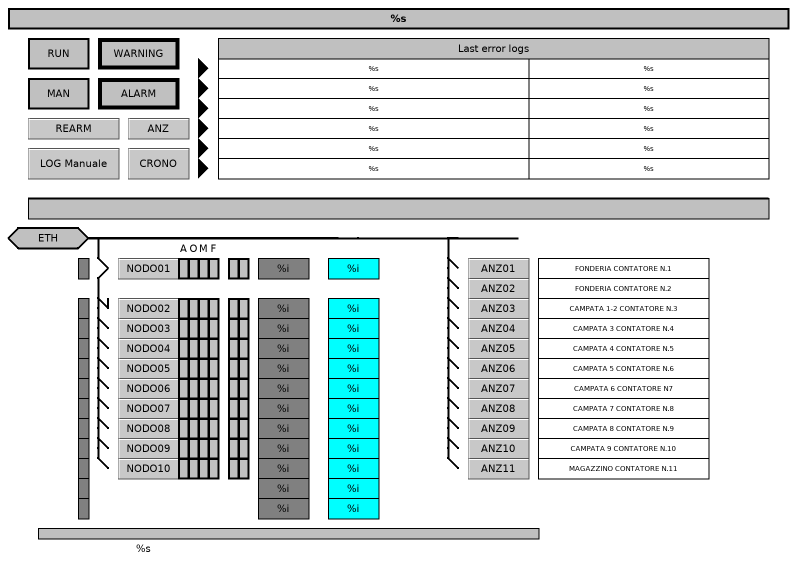
rectangle at (10,0)-(791,21): text "%s"; shows .Plant_NAME
rounded rectangle at (30,30)-(91,61): text "RUN"; alarm colour if NOT Mode_Manual; runs INTERN ASSIGN Mode_Manual:=(FALSE)
rounded rectangle at (30,70)-(91,101): text "MAN"; alarm colour if Mode_Manual; runs INTERN ASSIGN Mode_Manual:=(TRUE)
rectangle at (530,50)-(771,71): text "%s"; shows Sys.LastLogs_Msg[0]
polygon at (200,150)-(210,170): invisible if Sys.LastLogs_Idx<>0
rectangle at (530,70)-(771,91): text "%s"; shows Sys.LastLogs_Msg[1]
polygon at (200,50)-(210,70): invisible if Sys.LastLogs_Idx<>1
rectangle at (530,90)-(771,111): text "%s"; shows Sys.LastLogs_Msg[2]
polygon at (200,70)-(210,90): invisible if Sys.LastLogs_Idx<>2
rectangle at (530,110)-(771,131): text "%s"; shows Sys.LastLogs_Msg[3]
polygon at (200,90)-(210,110): invisible if Sys.LastLogs_Idx<>3
rectangle at (530,130)-(771,151): text "%s"; shows Sys.LastLogs_Msg[4]
polygon at (200,110)-(210,130): invisible if Sys.LastLogs_Idx<>4
rectangle at (530,150)-(771,171): text "%s"; shows Sys.LastLogs_Msg[5]
polygon at (200,130)-(210,150): invisible if Sys.LastLogs_Idx<>5
rectangle at (220,50)-(531,71): text "%s"; shows Sys.LastLogs_Dat[0]
rectangle at (220,70)-(531,91): text "%s"; shows Sys.LastLogs_Dat[1]
rectangle at (220,90)-(531,111): text "%s"; shows Sys.LastLogs_Dat[2]
rectangle at (220,110)-(531,131): text "%s"; shows Sys.LastLogs_Dat[3]
rectangle at (220,130)-(531,151): text "%s"; shows Sys.LastLogs_Dat[4]
rectangle at (220,150)-(531,171): text "%s"; shows Sys.LastLogs_Dat[5]
rectangle at (100,70)-(181,101): text "ALARM"; alarm colour if Sys.Alarm; runs INTERN ASSIGN Mode_Manual:=(FALSE)
rectangle at (100,30)-(181,61): text "WARNING"; alarm colour if Sys.Warning; runs INTERN ASSIGN Mode_Manual:=(TRUE)
button at (30,110)-(121,131): text "REARM"; runs INTERN ASSIGN Sys.Alarm:=(FALSE);INTERN ASSIGN Sys.Warning:=(FALSE)
button at (470,250)-(531,271): text "ANZ01"
rectangle at (220,30)-(771,51): text "Last error logs"
button at (470,270)-(531,291): text "ANZ02"
rectangle at (40,530)-(251,551): text "%s"; shows Sys.Time_LogString
button at (470,290)-(531,311): text "ANZ03"
button at (470,310)-(531,331): text "ANZ04"
button at (470,330)-(531,351): text "ANZ05"
button at (30,140)-(121,171): text "LOG Manuale"; taps PLC_PRG.HMI_AggiornaLog
polygon at (10,220)-(90,240): text "ETH"
button at (470,350)-(531,371): text "ANZ06"
button at (470,370)-(531,391): text "ANZ07"
button at (470,390)-(531,411): text "ANZ08"
button at (470,410)-(531,431): text "ANZ09"
button at (470,430)-(531,451): text "ANZ10"
button at (470,450)-(531,471): text "ANZ11"
button at (120,250)-(181,271): text "NODO01"
rectangle at (180,250)-(191,271): alarm colour if .NODO01.DI_01
rectangle at (190,250)-(201,271): alarm colour if .NODO01.DI_02
rectangle at (200,250)-(211,271): alarm colour if .NODO01.DI_03
rectangle at (210,250)-(221,271): alarm colour if .NODO01.DI_04
button at (120,290)-(181,311): text "NODO02"
rectangle at (180,290)-(191,311): alarm colour if .NODO02.DI_01
rectangle at (190,290)-(201,311): alarm colour if .NODO02.DI_02
rectangle at (200,290)-(211,311): alarm colour if .NODO02.DI_03
rectangle at (210,290)-(221,311): alarm colour if .NODO02.DI_04
button at (120,310)-(181,331): text "NODO03"
rectangle at (180,310)-(191,331): alarm colour if .NODO03.DI_01
rectangle at (190,310)-(201,331): alarm colour if .NODO03.DI_02
rectangle at (200,310)-(211,331): alarm colour if .NODO03.DI_03
rectangle at (210,310)-(221,331): alarm colour if .NODO03.DI_04
button at (120,330)-(181,351): text "NODO04"
rectangle at (180,330)-(191,351): alarm colour if .NODO04.DI_01
rectangle at (190,330)-(201,351): alarm colour if .NODO04.DI_02
rectangle at (200,330)-(211,351): alarm colour if .NODO04.DI_03
rectangle at (210,330)-(221,351): alarm colour if .NODO04.DI_04
button at (120,350)-(181,371): text "NODO05"
rectangle at (180,350)-(191,371): alarm colour if .NODO05.DI_01
rectangle at (190,350)-(201,371): alarm colour if .NODO05.DI_02
rectangle at (200,350)-(211,371): alarm colour if .NODO05.DI_03
rectangle at (210,350)-(221,371): alarm colour if .NODO05.DI_04
button at (120,370)-(181,391): text "NODO06"
rectangle at (180,370)-(191,391): alarm colour if .NODO06.DI_01
rectangle at (190,370)-(201,391): alarm colour if .NODO06.DI_02
rectangle at (200,370)-(211,391): alarm colour if .NODO06.DI_03
rectangle at (210,370)-(221,391): alarm colour if .NODO06.DI_04
button at (120,390)-(181,411): text "NODO07"
rectangle at (180,390)-(191,411): alarm colour if .NODO07.DI_01
rectangle at (190,390)-(201,411): alarm colour if .NODO07.DI_02
rectangle at (200,390)-(211,411): alarm colour if .NODO07.DI_03
rectangle at (210,390)-(221,411): alarm colour if .NODO07.DI_04
button at (120,410)-(181,431): text "NODO08"
rectangle at (180,410)-(191,431): alarm colour if .NODO08.DI_01
rectangle at (190,410)-(201,431): alarm colour if .NODO08.DI_02
rectangle at (200,410)-(211,431): alarm colour if .NODO08.DI_03
rectangle at (210,410)-(221,431): alarm colour if .NODO08.DI_04
button at (120,430)-(181,451): text "NODO09"
rectangle at (180,430)-(191,451): alarm colour if .NODO09.DI_01
rectangle at (190,430)-(201,451): alarm colour if .NODO09.DI_02
rectangle at (200,430)-(211,451): alarm colour if .NODO09.DI_03
rectangle at (210,430)-(221,451): alarm colour if .NODO09.DI_04
button at (120,450)-(181,471): text "NODO10"
rectangle at (180,450)-(191,471): alarm colour if .NODO10.DI_01
rectangle at (190,450)-(201,471): alarm colour if .NODO10.DI_02
rectangle at (200,450)-(211,471): alarm colour if .NODO10.DI_03
rectangle at (210,450)-(221,471): alarm colour if .NODO10.DI_04
rectangle at (230,250)-(241,271): alarm colour if .NODO01.DO_01
rectangle at (240,250)-(251,271): alarm colour if .NODO01.DO_02
rectangle at (230,290)-(241,311): alarm colour if .NODO02.DO_01
rectangle at (240,290)-(251,311): alarm colour if .NODO02.DO_02
rectangle at (230,310)-(241,331): alarm colour if .NODO03.DO_01
rectangle at (240,310)-(251,331): alarm colour if .NODO03.DO_02
rectangle at (230,330)-(241,351): alarm colour if .NODO04.DO_01
rectangle at (240,330)-(251,351): alarm colour if .NODO04.DO_02
rectangle at (230,350)-(241,371): alarm colour if .NODO05.DO_01
rectangle at (240,350)-(251,371): alarm colour if .NODO05.DO_02
rectangle at (230,370)-(241,391): alarm colour if .NODO06.DO_01
rectangle at (240,370)-(251,391): alarm colour if .NODO06.DO_02
rectangle at (230,390)-(241,411): alarm colour if .NODO07.DO_01
rectangle at (240,390)-(251,411): alarm colour if .NODO07.DO_02
rectangle at (230,410)-(241,431): alarm colour if .NODO08.DO_01
rectangle at (240,410)-(251,431): alarm colour if .NODO08.DO_02
rectangle at (230,430)-(241,451): alarm colour if .NODO09.DO_01
rectangle at (240,430)-(251,451): alarm colour if .NODO09.DO_02
rectangle at (230,450)-(241,471): alarm colour if .NODO10.DO_01
rectangle at (240,450)-(251,471): alarm colour if .NODO10.DO_02
rectangle at (540,250)-(711,271): text "FONDERIA CONTATORE N.1"
rectangle at (540,270)-(711,291): text "FONDERIA CONTATORE N.2"
rectangle at (540,290)-(711,311): text "CAMPATA 1-2 CONTATORE N.3"
rectangle at (540,310)-(711,331): text "CAMPATA 3 CONTATORE N.4"
rectangle at (540,330)-(711,351): text "CAMPATA 4 CONTATORE N.5"
rectangle at (540,350)-(711,371): text "CAMPATA 5 CONTATORE N.6"
rectangle at (540,370)-(711,391): text "CAMPATA 6 CONTATORE N7"
rectangle at (540,390)-(711,411): text "CAMPATA 7 CONTATORE N.8"
rectangle at (540,410)-(711,431): text "CAMPATA 8 CONTATORE N.9"
rectangle at (540,430)-(711,451): text "CAMPATA 9 CONTATORE N.10"
rectangle at (540,450)-(711,471): text "MAGAZZINO CONTATORE N.11"
rectangle at (180,230)-(191,251): text "A"
rectangle at (190,230)-(201,251): text "O"
rectangle at (200,230)-(211,251): text "M"
rectangle at (210,230)-(221,251): text "F"
button at (130,140)-(191,171): text "CRONO"; opens VIS_CHONOEDITOR
rectangle at (80,250)-(91,271): alarm colour if .LuxElement01.Lux_Enable
rectangle at (80,290)-(91,311): alarm colour if .LuxElement02.Lux_Enable
rectangle at (80,310)-(91,331): alarm colour if .LuxElement03.Lux_Enable
rectangle at (80,330)-(91,351): alarm colour if .LuxElement04.Lux_Enable
rectangle at (80,350)-(91,371): alarm colour if .LuxElement05.Lux_Enable
rectangle at (80,370)-(91,391): alarm colour if .LuxElement06.Lux_Enable
rectangle at (80,390)-(91,411): alarm colour if .LuxElement07.Lux_Enable
rectangle at (80,410)-(91,431): alarm colour if .LuxElement08.Lux_Enable
rectangle at (80,430)-(91,451): alarm colour if .LuxElement09.Lux_Enable
rectangle at (80,450)-(91,471): alarm colour if .LuxElement10.Lux_Enable
rectangle at (80,470)-(91,491): alarm colour if .LuxElement11.Lux_Enable
rectangle at (80,490)-(91,511): alarm colour if .LuxElement12.Lux_Enable
rectangle at (260,250)-(311,271): text "%i"; shows .ZTHL01.ValoreScalato
rectangle at (260,290)-(311,311): text "%i"; shows .ZTHL02.ValoreScalato
rectangle at (260,310)-(311,331): text "%i"; shows .ZTHL03.ValoreScalato
rectangle at (260,330)-(311,351): text "%i"; shows .ZTHL04.ValoreScalato
rectangle at (260,350)-(311,371): text "%i"; shows .ZTHL05.ValoreScalato
rectangle at (260,370)-(311,391): text "%i"; shows .ZTHL06.ValoreScalato
rectangle at (260,390)-(311,411): text "%i"; shows .ZTHL07.ValoreScalato
rectangle at (260,410)-(311,431): text "%i"; shows .ZTHL08.ValoreScalato
rectangle at (260,430)-(311,451): text "%i"; shows .ZTHL09.ValoreScalato
rectangle at (260,450)-(311,471): text "%i"; shows .ZTHL10.ValoreScalato
button at (130,110)-(191,131): text "ANZ"; opens Vis_ANZ
rectangle at (330,250)-(381,271): text "%i"; shows PLC_PRG.SogliaLux01
rectangle at (330,290)-(381,311): text "%i"; shows PLC_PRG.SogliaLux02
rectangle at (330,310)-(381,331): text "%i"; shows PLC_PRG.SogliaLux03
rectangle at (330,330)-(381,351): text "%i"; shows PLC_PRG.SogliaLux04
rectangle at (330,350)-(381,371): text "%i"; shows PLC_PRG.SogliaLux05
rectangle at (330,370)-(381,391): text "%i"; shows PLC_PRG.SogliaLux06
rectangle at (330,390)-(381,411): text "%i"; shows PLC_PRG.SogliaLux07
rectangle at (330,410)-(381,431): text "%i"; shows PLC_PRG.SogliaLux08
rectangle at (330,430)-(381,451): text "%i"; shows PLC_PRG.SogliaLux09
rectangle at (330,450)-(381,471): text "%i"; shows PLC_PRG.SogliaLux10
rectangle at (260,470)-(311,491): text "%i"; shows .ZTHL02.ValoreScalato
rectangle at (260,490)-(311,511): text "%i"; shows .ZTHL03.ValoreScalato
rectangle at (330,470)-(381,491): text "%i"; shows PLC_PRG.SogliaLux11
rectangle at (330,490)-(381,511): text "%i"; shows PLC_PRG.SogliaLux12
25 more shapes without text or variables
33 elements of other kinds (tables, trends, ...) not read
*)

(* Visualisation Vis_ANZ
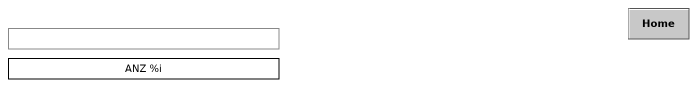
rectangle at (100,60)-(371,81): text "ANZ %i"; shows PLC_PRG.IndiceAnz
button at (720,10)-(781,41): text "Home"; opens PLC_VISU
1 more shapes without text or variables
1 elements of other kinds (tables, trends, ...) not read
*)

